LIN {X 0,Y 269.513,Z 759.84,A -85,B 0,C 180,E1 -29388.002,E2 -29388.002} C_VEL
LIN {X 0,Y 275.848,Z 764.701,A -85,B 0,C 180,E1 -29390.437,E2 -29390.437} C_VEL
LIN {X 0,Y 281.948,Z 769.462,A -85,B 0,C 180,E1 -29392.905,E2 -29392.905} C_VEL
LIN {X 0,Y 289.279,Z 774.875,A -85,B 0,C 180,E1 -29396.029,E2 -29396.029} C_VEL
LIN {X 0,Y 294.079,Z 778.705,A -85,B 0,C 180,E1 -29398.281,E2 -29398.281} C_VEL
LIN {X 0,Y 298.716,Z 782.114,A -85,B 0,C 180,E1 -29400.517,E2 -29400.517} C_VEL
LIN {X 0,Y 303.536,Z 785.554,A -85,B 0,C 180,E1 -29402.995,E2 -29402.995} C_VEL
LIN {X 0,Y 308.5,Z 789.254,A -85,B 0,C 180,E1 -29405.792,E2 -29405.792} C_VEL
LIN {X 0,Y 311.598,Z 791.295,A -85,B 0,C 180,E1 -29407.628,E2 -29407.628} C_VEL
LIN {X 0,Y 314.778,Z 793.373,A -85,B 0,C 180,E1 -29409.672,E2 -29409.672} C_VEL
LIN {X 0,Y 317.869,Z 795.742,A -85,B 0,C 180,E1 -29411.969,E2 -29411.969} C_VEL
LIN {X 0,Y 321.084,Z 798.198,A -85,B 0,C 180,E1 -29414.772,E2 -29414.772} C_VEL
LIN {X 0,Y 323.911,Z 800.084,A -85,B 0,C 180,E1 -29417.519,E2 -29417.519} C_VEL
LIN {X 0,Y 326.293,Z 801.22,A -85,B 0,C 180,E1 -29420.078,E2 -29420.078} C_VEL
LIN {X 0,Y 328.105,Z 802.015,A -85,B 0,C 180,E1 -29422.616,E2 -29422.616} C_VEL
LIN {X 0,Y 329.27,Z 802.725,A -85,B 0,C 180,E1 -29425.102,E2 -29425.102} C_VEL
LIN {X 0,Y 330.146,Z 802.967,A -85,B 0,C 180,E1 -29427.56,E2 -29427.56} C_VEL
LIN {X 0,Y 330.328,Z 803.159,A -85,B 0,C 180,E1 -29430,E2 -29430} C_VEL
LIN {X 0,Y 330.117,Z 802.967,A -85,B 0,C 180,E1 -29432.44,E2 -29432.44} C_VEL
LIN {X 0,Y 329.312,Z 802.689,A -85,B 0,C 180,E1 -29434.897,E2 -29434.897} C_VEL
LIN {X 0,Y 328.123,Z 802.039,A -85,B 0,C 180,E1 -29437.383,E2 -29437.383} C_VEL
LIN {X 0,Y 326.265,Z 801.233,A -85,B 0,C 180,E1 -29439.923,E2 -29439.923} C_VEL
LIN {X 0,Y 323.871,Z 800.004,A -85,B 0,C 180,E1 -29442.533,E2 -29442.533} C_VEL
LIN {X 0,Y 320.809,Z 798.053,A -85,B 0,C 180,E1 -29445.442,E2 -29445.442} C_VEL
LIN {X 0,Y 317.814,Z 795.774,A -85,B 0,C 180,E1 -29448.034,E2 -29448.034} C_VEL
LIN {X 0,Y 314.765,Z 793.38,A -85,B 0,C 180,E1 -29450.322,E2 -29450.322} C_VEL
LIN {X 0,Y 311.247,Z 791.126,A -85,B 0,C 180,E1 -29452.573,E2 -29452.573} C_VEL
LIN {X 0,Y 305.558,Z 787.096,A -85,B 0,C 180,E1 -29455.913,E2 -29455.913} C_VEL
LIN {X 0,Y 300.069,Z 782.993,A -85,B 0,C 180,E1 -29458.828,E2 -29458.828} C_VEL
LIN {X 0,Y 294.071,Z 778.695,A -85,B 0,C 180,E1 -29461.72,E2 -29461.72} C_VEL
LIN {X 0,Y 288.811,Z 774.531,A -85,B 0,C 180,E1 -29464.172,E2 -29464.172} C_VEL
LIN {X 0,Y 281.952,Z 769.478,A -85,B 0,C 180,E1 -29467.096,E2 -29467.096} C_VEL
LIN {X 0,Y 275.891,Z 764.765,A -85,B 0,C 180,E1 -29469.556,E2 -29469.556} C_VEL
LIN {X 0,Y 269.548,Z 759.774,A -85,B 0,C 180,E1 -29472.006,E2 -29472.006} C_VEL
LIN {X 0,Y 260.297,Z 752.713,A -85,B 0,C 180,E1 -29475.413,E2 -29475.413} C_VEL
LIN {X 0,Y 246.486,Z 741.482,A -85,B 0,C 180,E1 -29481.151,E2 -29481.151} C_VEL
LIN {X 0,Y 233.507,Z 728.442,A -85,B 0,C 180,E1 -29488.217,E2 -29488.217} C_VEL
LIN {X 0,Y 225.035,Z 716.362,A -85,B 0,C 180,E1 -29494.682,E2 -29494.682} C_VEL
LIN {X 0,Y 219.674,Z 703.721,A -85,B 0,C 180,E1 -29500.918,E2 -29500.918} C_VEL
LIN {X 0,Y 216.948,Z 692.283,A -85,B 0,C 180,E1 -29506.06,E2 -29506.06} C_VEL
LIN {X 0,Y 215.599,Z 681.886,A -85,B 0,C 180,E1 -29510.507,E2 -29510.507} C_VEL
LIN {X 0,Y 214.994,Z 678.195,A -85,B 0,C 180,E1 -29512.664,E2 -29512.664} C_VEL
LIN {X 0,Y 214.461,Z 674.849,A -85,B 0,C 180,E1 -29515.412,E2 -29515.412} C_VEL
LIN {X 0,Y 214.209,Z 673.133,A -85,B 0,C 180,E1 -29517.65,E2 -29517.65} C_VEL
LIN {X 0,Y 214.12,Z 672.763,A -85,B 0,C 180,E1 -29520.476,E2 -29520.476} C_VEL
LIN {X 0,Y 211.138,Z 691.221,A -85,B 0,C 180,E1 -29520.708,E2 -29520.708} C_VEL
LIN {X 0,Y 207.685,Z 705.637,A -85,B 0,C 180,E1 -29520.907,E2 -29520.907} C_VEL
LIN {X 0,Y 203.406,Z 719.374,A -85,B 0,C 180,E1 -29521.115,E2 -29521.115} C_VEL
LIN {X 0,Y 198.594,Z 731.963,A -85,B 0,C 180,E1 -29521.377,E2 -29521.377} C_VEL
LIN {X 0,Y 193.349,Z 743.558,A -85,B 0,C 180,E1 -29521.688,E2 -29521.688} C_VEL
LIN {X 0,Y 186.937,Z 755.704,A -85,B 0,C 180,E1 -29522.084,E2 -29522.084} C_VEL
LIN {X 0,Y 179.399,Z 768.002,A -85,B 0,C 180,E1 -29522.63,E2 -29522.63} C_VEL
LIN {X 0,Y 171.572,Z 779.121,A -85,B 0,C 180,E1 -29523.206,E2 -29523.206} C_VEL
LIN {X 0,Y 162.906,Z 789.948,A -85,B 0,C 180,E1 -29523.954,E2 -29523.954} C_VEL
LIN {X 0,Y 153.235,Z 800.571,A -85,B 0,C 180,E1 -29524.879,E2 -29524.879} C_VEL
LIN {X 0,Y 144.516,Z 809.109,A -85,B 0,C 180,E1 -29525.913,E2 -29525.913} C_VEL
LIN {X 0,Y 134.582,Z 817.767,A -85,B 0,C 180,E1 -29527.172,E2 -29527.172} C_VEL
LIN {X 0,Y 124.423,Z 825.65,A -85,B 0,C 180,E1 -29528.714,E2 -29528.714} C_VEL
LIN {X 0,Y 113.699,Z 833.04,A -85,B 0,C 180,E1 -29530.687,E2 -29530.687} C_VEL
LIN {X 0,Y 101.25,Z 840.568,A -85,B 0,C 180,E1 -29533.65,E2 -29533.65} C_VEL
LIN {X 0,Y 91.621,Z 845.7,A -85,B 0,C 180,E1 -29536.501,E2 -29536.501} C_VEL
LIN {X 0,Y 79.232,Z 851.465,A -85,B 0,C 180,E1 -29541.354,E2 -29541.354} C_VEL
LIN {X 0,Y 70.415,Z 855.088,A -85,B 0,C 180,E1 -29546.071,E2 -29546.071} C_VEL
LIN {X 0,Y 59.652,Z 858.961,A -85,B 0,C 180,E1 -29554.442,E2 -29554.442} C_VEL
LIN {X 0,Y 50.575,Z 861.84,A -85,B 0,C 180,E1 -29565.99,E2 -29565.99} C_VEL
LIN {X 0,Y 44.024,Z 863.755,A -85,B 0,C 180,E1 -29581.386,E2 -29581.386} C_VEL
LIN {X 0,Y 42.132,Z 864.451,A -85,B 0,C 180,E1 -29590.512,E2 -29590.512} C_VEL
LIN {X 0,Y 41.238,Z 864.959,A -85,B 0,C 180,E1 -29610,E2 -29610} C_VEL
LIN {X 0,Y 42.12,Z 864.45,A -85,B 0,C 180,E1 -29629.494,E2 -29629.494} C_VEL
LIN {X 0,Y 46.907,Z 862.99,A -85,B 0,C 180,E1 -29646.82,E2 -29646.82} C_VEL
LIN {X 0,Y 54.867,Z 860.576,A -85,B 0,C 180,E1 -29660.223,E2 -29660.223} C_VEL
LIN {X 0,Y 67.596,Z 856.132,A -85,B 0,C 180,E1 -29672.096,E2 -29672.096} C_VEL
LIN {X 0,Y 76.226,Z 852.753,A -85,B 0,C 180,E1 -29677.216,E2 -29677.216} C_VEL
LIN {X 0,Y 88.465,Z 847.245,A -85,B 0,C 180,E1 -29682.422,E2 -29682.422} C_VEL
LIN {X 0,Y 98.02,Z 842.385,A -85,B 0,C 180,E1 -29685.448,E2 -29685.448} C_VEL
LIN {X 0,Y 110.913,Z 834.823,A -85,B 0,C 180,E1 -29688.675,E2 -29688.675} C_VEL
LIN {X 0,Y 121.061,Z 828.065,A -85,B 0,C 180,E1 -29690.711,E2 -29690.711} C_VEL
LIN {X 0,Y 131.176,Z 820.52,A -85,B 0,C 180,E1 -29692.371,E2 -29692.371} C_VEL
LIN {X 0,Y 141.415,Z 811.951,A -85,B 0,C 180,E1 -29693.685,E2 -29693.685} C_VEL
LIN {X 0,Y 151.346,Z 802.524,A -85,B 0,C 180,E1 -29694.899,E2 -29694.899} C_VEL
LIN {X 0,Y 161.169,Z 791.956,A -85,B 0,C 180,E1 -29695.927,E2 -29695.927} C_VEL
LIN {X 0,Y 169.832,Z 781.404,A -85,B 0,C 180,E1 -29696.676,E2 -29696.676} C_VEL
LIN {X 0,Y 177.659,Z 770.609,A -85,B 0,C 180,E1 -29697.242,E2 -29697.242} C_VEL
LIN {X 0,Y 185.055,Z 758.937,A -85,B 0,C 180,E1 -29697.793,E2 -29697.793} C_VEL
LIN {X 0,Y 191.601,Z 747.036,A -85,B 0,C 180,E1 -29698.219,E2 -29698.219} C_VEL
LIN {X 0,Y 197.282,Z 735.038,A -85,B 0,C 180,E1 -29698.545,E2 -29698.545} C_VEL
LIN {X 0,Y 202.532,Z 721.843,A -85,B 0,C 180,E1 -29698.826,E2 -29698.826} C_VEL
LIN {X 0,Y 206.767,Z 708.849,A -85,B 0,C 180,E1 -29699.043,E2 -29699.043} C_VEL
LIN {X 0,Y 210.248,Z 695.285,A -85,B 0,C 180,E1 -29699.228,E2 -29699.228} C_VEL
LIN {X 0,Y 212.638,Z 682.821,A -85,B 0,C 180,E1 -29699.413,E2 -29699.413} C_VEL
LIN {X 0,Y 214.121,Z 672.732,A -85,B 0,C 180,E1 -29699.584,E2 -29699.584} C_VEL
LIN {X 0,Y 214.238,Z 673.333,A -85,B 0,C 180,E1 -29702.702,E2 -29702.702} C_VEL
LIN {X 0,Y 214.62,Z 675.963,A -85,B 0,C 180,E1 -29705.637,E2 -29705.637} C_VEL
LIN {X 0,Y 215.251,Z 679.856,A -85,B 0,C 180,E1 -29708.419,E2 -29708.419} C_VEL
LIN {X 0,Y 215.918,Z 684.51,A -85,B 0,C 180,E1 -29710.668,E2 -29710.668} C_VEL
LIN {X 0,Y 216.528,Z 689.348,A -85,B 0,C 180,E1 -29712.698,E2 -29712.698} C_VEL
LIN {X 0,Y 216.824,Z 691.412,A -85,B 0,C 180,E1 -29713.574,E2 -29713.574} C_VEL
LIN {X 0,Y 217.026,Z 695.327,A -85,B 0,C 180,E1 -29714.74,E2 -29714.74} C_VEL
LIN {X 0,Y 216.849,Z 707.033,A -85,B 0,C 180,E1 -29717.584,E2 -29717.584} C_VEL
LIN {X 0,Y 217.221,Z 710.631,A -85,B 0,C 180,E1 -29718.824,E2 -29718.824} C_VEL
LIN {X 0,Y 222.051,Z 722.799,A -85,B 0,C 180,E1 -29725.068,E2 -29725.068} C_VEL
LIN {X 0,Y 230.801,Z 735.633,A -85,B 0,C 180,E1 -29732.2,E2 -29732.2} C_VEL
LIN {X 0,Y 245.264,Z 749.741,A -85,B 0,C 180,E1 -29740.145,E2 -29740.145} C_VEL
LIN {X 0,Y 257.353,Z 759.43,A -85,B 0,C 180,E1 -29745.236,E2 -29745.236} C_VEL
LIN {X 0,Y 264.757,Z 765.09,A -85,B 0,C 180,E1 -29748.009,E2 -29748.009} C_VEL
LIN {X 0,Y 271.997,Z 770.662,A -85,B 0,C 180,E1 -29750.818,E2 -29750.818} C_VEL
LIN {X 0,Y 277.29,Z 774.8,A -85,B 0,C 180,E1 -29752.973,E2 -29752.973} C_VEL
LIN {X 0,Y 284.234,Z 779.942,A -85,B 0,C 180,E1 -29755.926,E2 -29755.926} C_VEL
LIN {X 0,Y 289.243,Z 783.893,A -85,B 0,C 180,E1 -29758.257,E2 -29758.257} C_VEL
LIN {X 0,Y 294.145,Z 787.523,A -85,B 0,C 180,E1 -29760.628,E2 -29760.628} C_VEL
LIN {X 0,Y 299.172,Z 791.122,A -85,B 0,C 180,E1 -29763.21,E2 -29763.21} C_VEL
LIN {X 0,Y 302.926,Z 793.936,A -85,B 0,C 180,E1 -29765.317,E2 -29765.317} C_VEL
LIN {X 0,Y 305.799,Z 795.921,A -85,B 0,C 180,E1 -29767.002,E2 -29767.002} C_VEL
LIN {X 0,Y 308.863,Z 797.869,A -85,B 0,C 180,E1 -29768.894,E2 -29768.894} C_VEL
LIN {X 0,Y 312.723,Z 800.732,A -85,B 0,C 180,E1 -29771.662,E2 -29771.662} C_VEL
LIN {X 0,Y 316.06,Z 803.297,A -85,B 0,C 180,E1 -29774.524,E2 -29774.524} C_VEL
LIN {X 0,Y 318.94,Z 805.266,A -85,B 0,C 180,E1 -29777.27,E2 -29777.27} C_VEL
LIN {X 0,Y 321.428,Z 806.457,A -85,B 0,C 180,E1 -29779.926,E2 -29779.926} C_VEL
LIN {X 0,Y 323.337,Z 807.296,A -85,B 0,C 180,E1 -29782.507,E2 -29782.507} C_VEL
LIN {X 0,Y 324.551,Z 808.043,A -85,B 0,C 180,E1 -29785.031,E2 -29785.031} C_VEL
LIN {X 0,Y 325.474,Z 808.31,A -85,B 0,C 180,E1 -29787.525,E2 -29787.525} C_VEL
LIN {X 0,Y 325.699,Z 808.396,A -85,B 0,C 180,E1 -29788.764,E2 -29788.764} C_VEL
LIN {X 0,Y 325.626,Z 808.426,A -85,B 0,C 180,E1 -29791.237,E2 -29791.237} C_VEL
LIN {X 0,Y 325.034,Z 808.243,A -85,B 0,C 180,E1 -29793.719,E2 -29793.719} C_VEL
LIN {X 0,Y 324.061,Z 807.683,A -85,B 0,C 180,E1 -29796.225,E2 -29796.225} C_VEL
LIN {X 0,Y 322.442,Z 806.929,A -85,B 0,C 180,E1 -29798.776,E2 -29798.776} C_VEL
LIN {X 0,Y 320.245,Z 805.898,A -85,B 0,C 180,E1 -29801.391,E2 -29801.391} C_VEL
LIN {X 0,Y 317.542,Z 804.326,A -85,B 0,C 180,E1 -29804.09,E2 -29804.09} C_VEL
LIN {X 0,Y 314.395,Z 802.115,A -85,B 0,C 180,E1 -29806.894,E2 -29806.894} C_VEL
LIN {X 0,Y 311.99,Z 800.188,A -85,B 0,C 180,E1 -29808.898,E2 -29808.898} C_VEL
LIN {X 0,Y 308.435,Z 797.598,A -85,B 0,C 180,E1 -29811.381,E2 -29811.381} C_VEL
LIN {X 0,Y 305.606,Z 795.851,A -85,B 0,C 180,E1 -29813.094,E2 -29813.094} C_VEL
LIN {X 0,Y 299.862,Z 791.627,A -85,B 0,C 180,E1 -29816.443,E2 -29816.443} C_VEL
LIN {X 0,Y 294.191,Z 787.506,A -85,B 0,C 180,E1 -29819.37,E2 -29819.37} C_VEL
LIN {X 0,Y 289.247,Z 783.903,A -85,B 0,C 180,E1 -29821.744,E2 -29821.744} C_VEL
LIN {X 0,Y 284.24,Z 779.944,A -85,B 0,C 180,E1 -29824.076,E2 -29824.076} C_VEL
LIN {X 0,Y 279.029,Z 776.124,A -85,B 0,C 180,E1 -29826.295,E2 -29826.295} C_VEL
LIN {X 0,Y 275.596,Z 773.373,A -85,B 0,C 180,E1 -29827.766,E2 -29827.766} C_VEL
LIN {X 0,Y 268.399,Z 767.914,A -85,B 0,C 180,E1 -29830.593,E2 -29830.593} C_VEL
LIN {X 0,Y 262.635,Z 763.36,A -85,B 0,C 180,E1 -29832.785,E2 -29832.785} C_VEL
LIN {X 0,Y 250.326,Z 753.803,A -85,B 0,C 180,E1 -29837.639,E2 -29837.639} C_VEL
LIN {X 0,Y 234.708,Z 740.007,A -85,B 0,C 180,E1 -29845.325,E2 -29845.325} C_VEL
LIN {X 0,Y 225.105,Z 728.004,A -85,B 0,C 180,E1 -29852.076,E2 -29852.076} C_VEL
LIN {X 0,Y 219.774,Z 718.027,A -85,B 0,C 180,E1 -29857.435,E2 -29857.435} C_VEL
LIN {X 0,Y 216.366,Z 707.28,A -85,B 0,C 180,E1 -29862.759,E2 -29862.759} C_VEL
LIN {X 0,Y 214.647,Z 696.607,A -85,B 0,C 180,E1 -29867.605,E2 -29867.605} C_VEL
LIN {X 0,Y 213.992,Z 687.722,A -85,B 0,C 180,E1 -29871.531,E2 -29871.531} C_VEL
LIN {X 0,Y 213.696,Z 684.84,A -85,B 0,C 180,E1 -29873.242,E2 -29873.242} C_VEL
LIN {X 0,Y 213.348,Z 681.75,A -85,B 0,C 180,E1 -29875.741,E2 -29875.741} C_VEL
LIN {X 0,Y 213.161,Z 680.078,A -85,B 0,C 180,E1 -29878.111,E2 -29878.111} C_VEL
LIN {X 0,Y 213.13,Z 679.974,A -85,B 0,C 180,E1 -29878.628,E2 -29878.628} C_VEL
LIN {X 0,Y 210.458,Z 694.251,A -85,B 0,C 180,E1 -29878.816,E2 -29878.816} C_VEL
LIN {X 0,Y 206.952,Z 708.017,A -85,B 0,C 180,E1 -29878.971,E2 -29878.971} C_VEL
LIN {X 0,Y 202.511,Z 721.639,A -85,B 0,C 180,E1 -29879.156,E2 -29879.156} C_VEL
LIN {X 0,Y 197.23,Z 734.836,A -85,B 0,C 180,E1 -29879.381,E2 -29879.381} C_VEL
LIN {X 0,Y 190.633,Z 748.57,A -85,B 0,C 180,E1 -29879.697,E2 -29879.697} C_VEL
LIN {X 0,Y 180.968,Z 765.188,A -85,B 0,C 180,E1 -29880.256,E2 -29880.256} C_VEL
LIN {X 0,Y 172.197,Z 777.773,A -85,B 0,C 180,E1 -29880.752,E2 -29880.752} C_VEL
LIN {X 0,Y 163.445,Z 788.736,A -85,B 0,C 180,E1 -29881.387,E2 -29881.387} C_VEL
LIN {X 0,Y 154.71,Z 798.412,A -85,B 0,C 180,E1 -29882.033,E2 -29882.033} C_VEL
LIN {X 0,Y 145.707,Z 807.315,A -85,B 0,C 180,E1 -29882.877,E2 -29882.877} C_VEL
LIN {X 0,Y 135.611,Z 816.181,A -85,B 0,C 180,E1 -29883.966,E2 -29883.966} C_VEL
LIN {X 0,Y 123.537,Z 825.437,A -85,B 0,C 180,E1 -29885.407,E2 -29885.407} C_VEL
LIN {X 0,Y 113.281,Z 832.397,A -85,B 0,C 180,E1 -29886.965,E2 -29886.965} C_VEL
LIN {X 0,Y 103.144,Z 838.537,A -85,B 0,C 180,E1 -29888.895,E2 -29888.895} C_VEL
LIN {X 0,Y 89.836,Z 845.486,A -85,B 0,C 180,E1 -29892.076,E2 -29892.076} C_VEL
LIN {X 0,Y 79.188,Z 850.32,A -85,B 0,C 180,E1 -29895.442,E2 -29895.442} C_VEL
LIN {X 0,Y 67.558,Z 854.875,A -85,B 0,C 180,E1 -29900.571,E2 -29900.571} C_VEL
LIN {X 0,Y 55.889,Z 858.747,A -85,B 0,C 180,E1 -29908.331,E2 -29908.331} C_VEL
LIN {X 0,Y 49.655,Z 860.644,A -85,B 0,C 180,E1 -29914.484,E2 -29914.484} C_VEL
LIN {X 0,Y 41.387,Z 862.778,A -85,B 0,C 180,E1 -29927.217,E2 -29927.217} C_VEL
LIN {X 0,Y 35.444,Z 864.239,A -85,B 0,C 180,E1 -29946.637,E2 -29946.637} C_VEL
LIN {X 0,Y 34.113,Z 864.748,A -85,B 0,C 180,E1 -29970,E2 -29970} C_VEL
LIN {X 0,Y 35.435,Z 864.238,A -85,B 0,C 180,E1 -29993.37,E2 -29993.37} C_VEL
LIN {X 0,Y 41.386,Z 862.778,A -85,B 0,C 180,E1 -30012.785,E2 -30012.785} C_VEL
LIN {X 0,Y 50.551,Z 860.362,A -85,B 0,C 180,E1 -30026.527,E2 -30026.527} C_VEL
LIN {X 0,Y 64.534,Z 855.919,A -85,B 0,C 180,E1 -30037.767,E2 -30037.767} C_VEL
LIN {X 0,Y 73.73,Z 852.54,A -85,B 0,C 180,E1 -30042.399,E2 -30042.399} C_VEL
LIN {X 0,Y 86.56,Z 847.032,A -85,B 0,C 180,E1 -30046.978,E2 -30046.978} C_VEL
LIN {X 0,Y 96.457,Z 842.171,A -85,B 0,C 180,E1 -30049.61,E2 -30049.61} C_VEL
LIN {X 0,Y 109.237,Z 834.915,A -85,B 0,C 180,E1 -30052.278,E2 -30052.278} C_VEL
LIN {X 0,Y 120.108,Z 827.852,A -85,B 0,C 180,E1 -30054.109,E2 -30054.109} C_VEL
LIN {X 0,Y 130.416,Z 820.307,A -85,B 0,C 180,E1 -30055.504,E2 -30055.504} C_VEL
LIN {X 0,Y 140.806,Z 811.74,A -85,B 0,C 180,E1 -30056.587,E2 -30056.587} C_VEL
LIN {X 0,Y 151.225,Z 801.959,A -85,B 0,C 180,E1 -30057.652,E2 -30057.652} C_VEL
LIN {X 0,Y 160.819,Z 791.748,A -85,B 0,C 180,E1 -30058.464,E2 -30058.464} C_VEL
LIN {X 0,Y 169.568,Z 781.199,A -85,B 0,C 180,E1 -30059.076,E2 -30059.076} C_VEL
LIN {X 0,Y 177.458,Z 770.402,A -85,B 0,C 180,E1 -30059.545,E2 -30059.545} C_VEL
LIN {X 0,Y 184.757,Z 759.006,A -85,B 0,C 180,E1 -30060,E2 -30060} C_VEL
LIN {X 0,Y 191.512,Z 746.83,A -85,B 0,C 180,E1 -30060.348,E2 -30060.348} C_VEL
LIN {X 0,Y 197.23,Z 734.836,A -85,B 0,C 180,E1 -30060.618,E2 -30060.618} C_VEL
LIN {X 0,Y 202.511,Z 721.64,A -85,B 0,C 180,E1 -30060.836,E2 -30060.836} C_VEL
LIN {X 0,Y 206.73,Z 708.788,A -85,B 0,C 180,E1 -30061.01,E2 -30061.01} C_VEL
LIN {X 0,Y 210.233,Z 695.271,A -85,B 0,C 180,E1 -30061.164,E2 -30061.164} C_VEL
LIN {X 0,Y 212.782,Z 681.98,A -85,B 0,C 180,E1 -30061.333,E2 -30061.333} C_VEL
LIN {X 0,Y 213.102,Z 679.928,A -85,B 0,C 180,E1 -30061.372,E2 -30061.372} C_VEL
LIN {X 0,Y 213.183,Z 680.8,A -85,B 0,C 180,E1 -30063.07,E2 -30063.07} C_VEL
LIN {X 0,Y 213.486,Z 683.323,A -85,B 0,C 180,E1 -30065.667,E2 -30065.667} C_VEL
LIN {X 0,Y 213.912,Z 686.53,A -85,B 0,C 180,E1 -30067.848,E2 -30067.848} C_VEL
LIN {X 0,Y 214.208,Z 691.624,A -85,B 0,C 180,E1 -30070.252,E2 -30070.252} C_VEL
LIN {X 0,Y 215.674,Z 704.072,A -85,B 0,C 180,E1 -30075.716,E2 -30075.716} C_VEL
LIN {X 0,Y 217.221,Z 710.631,A -85,B 0,C 180,E1 -30078.824,E2 -30078.824} C_VEL
LIN {X 0,Y 217.704,Z 714.076,A -85,B 0,C 180,E1 -30080.089,E2 -30080.089} C_VEL
LIN {X 0,Y 218.379,Z 727.051,A -85,B 0,C 180,E1 -30084.004,E2 -30084.004} C_VEL
LIN {X 0,Y 219.25,Z 729.971,A -85,B 0,C 180,E1 -30085.317,E2 -30085.317} C_VEL
LIN {X 0,Y 226.67,Z 741.194,A -85,B 0,C 180,E1 -30091.809,E2 -30091.809} C_VEL
LIN {X 0,Y 239.104,Z 753.74,A -85,B 0,C 180,E1 -30099.193,E2 -30099.193} C_VEL
LIN {X 0,Y 250.711,Z 763.192,A -85,B 0,C 180,E1 -30104.491,E2 -30104.491} C_VEL
LIN {X 0,Y 259.783,Z 770.151,A -85,B 0,C 180,E1 -30108.07,E2 -30108.07} C_VEL
LIN {X 0,Y 266.852,Z 775.583,A -85,B 0,C 180,E1 -30110.797,E2 -30110.797} C_VEL
LIN {X 0,Y 274.503,Z 781.5,A -85,B 0,C 180,E1 -30113.925,E2 -30113.925} C_VEL
LIN {X 0,Y 280.674,Z 786.071,A -85,B 0,C 180,E1 -30116.574,E2 -30116.574} C_VEL
LIN {X 0,Y 286.252,Z 790.444,A -85,B 0,C 180,E1 -30119.238,E2 -30119.238} C_VEL
LIN {X 0,Y 291.295,Z 794.06,A -85,B 0,C 180,E1 -30121.715,E2 -30121.715} C_VEL
LIN {X 0,Y 296.224,Z 797.714,A -85,B 0,C 180,E1 -30124.362,E2 -30124.362} C_VEL
LIN {X 0,Y 299.987,Z 800.438,A -85,B 0,C 180,E1 -30126.53,E2 -30126.53} C_VEL
LIN {X 0,Y 305.214,Z 803.872,A -85,B 0,C 180,E1 -30129.794,E2 -30129.794} C_VEL
LIN {X 0,Y 307.291,Z 805.44,A -85,B 0,C 180,E1 -30131.326,E2 -30131.326} C_VEL
LIN {X 0,Y 310.769,Z 808.143,A -85,B 0,C 180,E1 -30134.254,E2 -30134.254} C_VEL
LIN {X 0,Y 313.736,Z 810.196,A -85,B 0,C 180,E1 -30137.056,E2 -30137.056} C_VEL
LIN {X 0,Y 316.301,Z 811.474,A -85,B 0,C 180,E1 -30139.761,E2 -30139.761} C_VEL
LIN {X 0,Y 318.33,Z 812.356,A -85,B 0,C 180,E1 -30142.388,E2 -30142.388} C_VEL
LIN {X 0,Y 319.622,Z 813.123,A -85,B 0,C 180,E1 -30144.954,E2 -30144.954} C_VEL
LIN {X 0,Y 320.566,Z 813.433,A -85,B 0,C 180,E1 -30147.487,E2 -30147.487} C_VEL
LIN {X 0,Y 320.806,Z 813.51,A -85,B 0,C 180,E1 -30148.745,E2 -30148.745} C_VEL
LIN {X 0,Y 320.716,Z 813.556,A -85,B 0,C 180,E1 -30151.256,E2 -30151.256} C_VEL
LIN {X 0,Y 320.539,Z 813.431,A -85,B 0,C 180,E1 -30152.513,E2 -30152.513} C_VEL
LIN {X 0,Y 319.665,Z 813.099,A -85,B 0,C 180,E1 -30155.045,E2 -30155.045} C_VEL
LIN {X 0,Y 318.33,Z 812.397,A -85,B 0,C 180,E1 -30157.612,E2 -30157.612} C_VEL
LIN {X 0,Y 316.288,Z 811.464,A -85,B 0,C 180,E1 -30160.239,E2 -30160.239} C_VEL
LIN {X 0,Y 313.763,Z 810.131,A -85,B 0,C 180,E1 -30162.943,E2 -30162.943} C_VEL
LIN {X 0,Y 310.723,Z 808.146,A -85,B 0,C 180,E1 -30165.748,E2 -30165.748} C_VEL
LIN {X 0,Y 307.272,Z 805.442,A -85,B 0,C 180,E1 -30168.675,E2 -30168.675} C_VEL
LIN {X 0,Y 305.219,Z 803.889,A -85,B 0,C 180,E1 -30170.205,E2 -30170.205} C_VEL
LIN {X 0,Y 302.732,Z 802.227,A -85,B 0,C 180,E1 -30171.804,E2 -30171.804} C_VEL
LIN {X 0,Y 299.467,Z 800.127,A -85,B 0,C 180,E1 -30173.758,E2 -30173.758} C_VEL
LIN {X 0,Y 293.734,Z 795.821,A -85,B 0,C 180,E1 -30177.039,E2 -30177.039} C_VEL
LIN {X 0,Y 289.667,Z 792.874,A -85,B 0,C 180,E1 -30179.14,E2 -30179.14} C_VEL
LIN {X 0,Y 282.904,Z 787.825,A -85,B 0,C 180,E1 -30182.368,E2 -30182.368} C_VEL
LIN {X 0,Y 277.992,Z 784.082,A -85,B 0,C 180,E1 -30184.584,E2 -30184.584} C_VEL
LIN {X 0,Y 271.434,Z 779.106,A -85,B 0,C 180,E1 -30187.357,E2 -30187.357} C_VEL
LIN {X 0,Y 265.294,Z 774.465,A -85,B 0,C 180,E1 -30189.804,E2 -30189.804} C_VEL
LIN {X 0,Y 257.977,Z 768.668,A -85,B 0,C 180,E1 -30192.647,E2 -30192.647} C_VEL
LIN {X 0,Y 245.577,Z 759.11,A -85,B 0,C 180,E1 -30197.738,E2 -30197.738} C_VEL
LIN {X 0,Y 230.449,Z 745.541,A -85,B 0,C 180,E1 -30205.653,E2 -30205.653} C_VEL
LIN {X 0,Y 220.993,Z 733.049,A -85,B 0,C 180,E1 -30212.927,E2 -30212.927} C_VEL
LIN {X 0,Y 216.401,Z 723.37,A -85,B 0,C 180,E1 -30218.308,E2 -30218.308} C_VEL
LIN {X 0,Y 213.592,Z 712.701,A -85,B 0,C 180,E1 -30223.759,E2 -30223.759} C_VEL
LIN {X 0,Y 212.397,Z 700.51,A -85,B 0,C 180,E1 -30229.379,E2 -30229.379} C_VEL
LIN {X 0,Y 212.235,Z 693.67,A -85,B 0,C 180,E1 -30232.461,E2 -30232.461} C_VEL
LIN {X 0,Y 212.142,Z 691.135,A -85,B 0,C 180,E1 -30234.035,E2 -30234.035} C_VEL
LIN {X 0,Y 212.057,Z 688.368,A -85,B 0,C 180,E1 -30236.414,E2 -30236.414} C_VEL
LIN {X 0,Y 212.038,Z 688.086,A -85,B 0,C 180,E1 -30236.797,E2 -30236.797} C_VEL
LIN {X 0,Y 208.044,Z 704.898,A -85,B 0,C 180,E1 -30236.986,E2 -30236.986} C_VEL
LIN {X 0,Y 203.626,Z 718.969,A -85,B 0,C 180,E1 -30237.117,E2 -30237.117} C_VEL
LIN {X 0,Y 198.76,Z 731.56,A -85,B 0,C 180,E1 -30237.279,E2 -30237.279} C_VEL
LIN {X 0,Y 193.455,Z 743.145,A -85,B 0,C 180,E1 -30237.464,E2 -30237.464} C_VEL
LIN {X 0,Y 187.001,Z 755.229,A -85,B 0,C 180,E1 -30237.719,E2 -30237.719} C_VEL
LIN {X 0,Y 179.311,Z 767.588,A -85,B 0,C 180,E1 -30238.077,E2 -30238.077} C_VEL
LIN {X 0,Y 171.368,Z 778.709,A -85,B 0,C 180,E1 -30238.422,E2 -30238.422} C_VEL
LIN {X 0,Y 162.547,Z 789.533,A -85,B 0,C 180,E1 -30238.929,E2 -30238.929} C_VEL
LIN {X 0,Y 152.861,Z 799.977,A -85,B 0,C 180,E1 -30239.493,E2 -30239.493} C_VEL
LIN {X 0,Y 143.041,Z 809.317,A -85,B 0,C 180,E1 -30240.25,E2 -30240.25} C_VEL
LIN {X 0,Y 133.552,Z 817.349,A -85,B 0,C 180,E1 -30241.076,E2 -30241.076} C_VEL
LIN {X 0,Y 123.067,Z 825.227,A -85,B 0,C 180,E1 -30242.071,E2 -30242.071} C_VEL
LIN {X 0,Y 112.635,Z 832.186,A -85,B 0,C 180,E1 -30243.326,E2 -30243.326} C_VEL
LIN {X 0,Y 102.276,Z 838.324,A -85,B 0,C 180,E1 -30244.89,E2 -30244.89} C_VEL
LIN {X 0,Y 88.608,Z 845.273,A -85,B 0,C 180,E1 -30247.509,E2 -30247.509} C_VEL
LIN {X 0,Y 76.671,Z 850.458,A -85,B 0,C 180,E1 -30250.565,E2 -30250.565} C_VEL
LIN {X 0,Y 65.368,Z 854.661,A -85,B 0,C 180,E1 -30254.624,E2 -30254.624} C_VEL
LIN {X 0,Y 52.847,Z 858.534,A -85,B 0,C 180,E1 -30261.425,E2 -30261.425} C_VEL
LIN {X 0,Y 41.443,Z 861.414,A -85,B 0,C 180,E1 -30272.018,E2 -30272.018} C_VEL
LIN {X 0,Y 36.45,Z 862.566,A -85,B 0,C 180,E1 -30279.536,E2 -30279.536} C_VEL
LIN {X 0,Y 29.004,Z 864.027,A -85,B 0,C 180,E1 -30301.012,E2 -30301.012} C_VEL
LIN {X 0,Y 27.001,Z 864.538,A -85,B 0,C 180,E1 -30330,E2 -30330} C_VEL
LIN {X 0,Y 28.996,Z 864.026,A -85,B 0,C 180,E1 -30358.996,E2 -30358.996} C_VEL
LIN {X 0,Y 36.449,Z 862.566,A -85,B 0,C 180,E1 -30380.466,E2 -30380.466} C_VEL
LIN {X 0,Y 46.962,Z 860.149,A -85,B 0,C 180,E1 -30393.884,E2 -30393.884} C_VEL
LIN {X 0,Y 62.167,Z 855.706,A -85,B 0,C 180,E1 -30403.924,E2 -30403.924} C_VEL
LIN {X 0,Y 71.878,Z 852.326,A -85,B 0,C 180,E1 -30407.889,E2 -30407.889} C_VEL
LIN {X 0,Y 85.224,Z 846.819,A -85,B 0,C 180,E1 -30411.711,E2 -30411.711} C_VEL
LIN {X 0,Y 95.421,Z 841.958,A -85,B 0,C 180,E1 -30413.871,E2 -30413.871} C_VEL
LIN {X 0,Y 109.172,Z 834.295,A -85,B 0,C 180,E1 -30416.158,E2 -30416.158} C_VEL
LIN {X 0,Y 119.583,Z 827.641,A -85,B 0,C 180,E1 -30417.548,E2 -30417.548} C_VEL
LIN {X 0,Y 130.05,Z 820.099,A -85,B 0,C 180,E1 -30418.661,E2 -30418.661} C_VEL
LIN {X 0,Y 140.562,Z 811.531,A -85,B 0,C 180,E1 -30419.511,E2 -30419.511} C_VEL
LIN {X 0,Y 151.102,Z 801.751,A -85,B 0,C 180,E1 -30420.377,E2 -30420.377} C_VEL
LIN {X 0,Y 161.667,Z 790.536,A -85,B 0,C 180,E1 -30421.049,E2 -30421.049} C_VEL
LIN {X 0,Y 169.603,Z 780.994,A -85,B 0,C 180,E1 -30421.486,E2 -30421.486} C_VEL
LIN {X 0,Y 177.546,Z 770.195,A -85,B 0,C 180,E1 -30421.853,E2 -30421.853} C_VEL
LIN {X 0,Y 185.319,Z 758.081,A -85,B 0,C 180,E1 -30422.216,E2 -30422.216} C_VEL
LIN {X 0,Y 191.688,Z 746.624,A -85,B 0,C 180,E1 -30422.477,E2 -30422.477} C_VEL
LIN {X 0,Y 197.877,Z 733.609,A -85,B 0,C 180,E1 -30422.697,E2 -30422.697} C_VEL
LIN {X 0,Y 202.739,Z 721.437,A -85,B 0,C 180,E1 -30422.842,E2 -30422.842} C_VEL
LIN {X 0,Y 207.051,Z 708.334,A -85,B 0,C 180,E1 -30422.975,E2 -30422.975} C_VEL
LIN {X 0,Y 210.625,Z 694.501,A -85,B 0,C 180,E1 -30423.102,E2 -30423.102} C_VEL
LIN {X 0,Y 212.044,Z 688.072,A -85,B 0,C 180,E1 -30423.221,E2 -30423.221} C_VEL
LIN {X 0,Y 212.127,Z 690.643,A -85,B 0,C 180,E1 -30425.615,E2 -30425.615} C_VEL
LIN {X 0,Y 212.231,Z 693.397,A -85,B 0,C 180,E1 -30427.4,E2 -30427.4} C_VEL
LIN {X 0,Y 212.37,Z 699.837,A -85,B 0,C 180,E1 -30430.321,E2 -30430.321} C_VEL
LIN {X 0,Y 213.244,Z 710.724,A -85,B 0,C 180,E1 -30435.287,E2 -30435.287} C_VEL
LIN {X 0,Y 215.315,Z 720.217,A -85,B 0,C 180,E1 -30440.042,E2 -30440.042} C_VEL
LIN {X 0,Y 218.686,Z 728.888,A -85,B 0,C 180,E1 -30444.694,E2 -30444.694} C_VEL
LIN {X 0,Y 219.25,Z 729.971,A -85,B 0,C 180,E1 -30445.317,E2 -30445.317} C_VEL
LIN {X 0,Y 220.255,Z 732.871,A -85,B 0,C 180,E1 -30446.633,E2 -30446.633} C_VEL
LIN {X 0,Y 221.939,Z 744.931,A -85,B 0,C 180,E1 -30450.686,E2 -30450.686} C_VEL
LIN {X 0,Y 223.211,Z 747.668,A -85,B 0,C 180,E1 -30451.99,E2 -30451.99} C_VEL
LIN {X 0,Y 237.483,Z 761.727,A -85,B 0,C 180,E1 -30460.621,E2 -30460.621} C_VEL
LIN {X 0,Y 251.088,Z 772.326,A -85,B 0,C 180,E1 -30466.697,E2 -30466.697} C_VEL
LIN {X 0,Y 262.127,Z 780.772,A -85,B 0,C 180,E1 -30471.034,E2 -30471.034} C_VEL
LIN {X 0,Y 269.314,Z 786.352,A -85,B 0,C 180,E1 -30473.995,E2 -30473.995} C_VEL
LIN {X 0,Y 274.65,Z 790.301,A -85,B 0,C 180,E1 -30476.266,E2 -30476.266} C_VEL
LIN {X 0,Y 279.763,Z 794.297,A -85,B 0,C 180,E1 -30478.662,E2 -30478.662} C_VEL
LIN {X 0,Y 285.342,Z 798.361,A -85,B 0,C 180,E1 -30481.387,E2 -30481.387} C_VEL
LIN {X 0,Y 289.889,Z 801.706,A -85,B 0,C 180,E1 -30483.768,E2 -30483.768} C_VEL
LIN {X 0,Y 293.844,Z 804.616,A -85,B 0,C 180,E1 -30486.009,E2 -30486.009} C_VEL
LIN {X 0,Y 299.34,Z 808.275,A -85,B 0,C 180,E1 -30489.38,E2 -30489.38} C_VEL
LIN {X 0,Y 302.911,Z 810.928,A -85,B 0,C 180,E1 -30492.036,E2 -30492.036} C_VEL
LIN {X 0,Y 306.036,Z 813.295,A -85,B 0,C 180,E1 -30494.688,E2 -30494.688} C_VEL
LIN {X 0,Y 309.204,Z 815.381,A -85,B 0,C 180,E1 -30497.782,E2 -30497.782} C_VEL
LIN {X 0,Y 310.94,Z 816.24,A -85,B 0,C 180,E1 -30499.583,E2 -30499.583} C_VEL
LIN {X 0,Y 313.07,Z 817.204,A -85,B 0,C 180,E1 -30502.259,E2 -30502.259} C_VEL
LIN {X 0,Y 314.428,Z 817.965,A -85,B 0,C 180,E1 -30504.871,E2 -30504.871} C_VEL
LIN {X 0,Y 315.378,Z 818.273,A -85,B 0,C 180,E1 -30507.446,E2 -30507.446} C_VEL
LIN {X 0,Y 315.617,Z 818.363,A -85,B 0,C 180,E1 -30508.724,E2 -30508.724} C_VEL
LIN {X 0,Y 315.531,Z 818.398,A -85,B 0,C 180,E1 -30511.276,E2 -30511.276} C_VEL
LIN {X 0,Y 314.909,Z 818.202,A -85,B 0,C 180,E1 -30513.839,E2 -30513.839} C_VEL
LIN {X 0,Y 313.858,Z 817.638,A -85,B 0,C 180,E1 -30516.428,E2 -30516.428} C_VEL
LIN {X 0,Y 312.056,Z 816.792,A -85,B 0,C 180,E1 -30519.07,E2 -30519.07} C_VEL
LIN {X 0,Y 309.235,Z 815.353,A -85,B 0,C 180,E1 -30522.245,E2 -30522.245} C_VEL
LIN {X 0,Y 306.028,Z 813.333,A -85,B 0,C 180,E1 -30525.307,E2 -30525.307} C_VEL
LIN {X 0,Y 302.911,Z 810.962,A -85,B 0,C 180,E1 -30527.964,E2 -30527.964} C_VEL
LIN {X 0,Y 299.345,Z 808.302,A -85,B 0,C 180,E1 -30530.619,E2 -30530.619} C_VEL
LIN {X 0,Y 293.807,Z 804.62,A -85,B 0,C 180,E1 -30533.994,E2 -30533.994} C_VEL
LIN {X 0,Y 288.269,Z 800.479,A -85,B 0,C 180,E1 -30537.146,E2 -30537.146} C_VEL
LIN {X 0,Y 283.062,Z 796.723,A -85,B 0,C 180,E1 -30539.773,E2 -30539.773} C_VEL
LIN {X 0,Y 278.399,Z 793.216,A -85,B 0,C 180,E1 -30542.014,E2 -30542.014} C_VEL
LIN {X 0,Y 272.827,Z 788.956,A -85,B 0,C 180,E1 -30544.521,E2 -30544.521} C_VEL
LIN {X 0,Y 265.745,Z 783.57,A -85,B 0,C 180,E1 -30547.497,E2 -30547.497} C_VEL
LIN {X 0,Y 260.244,Z 779.401,A -85,B 0,C 180,E1 -30549.678,E2 -30549.678} C_VEL
LIN {X 0,Y 253.209,Z 773.845,A -85,B 0,C 180,E1 -30552.478,E2 -30552.478} C_VEL
LIN {X 0,Y 239.522,Z 763.409,A -85,B 0,C 180,E1 -30558.369,E2 -30558.369} C_VEL
LIN {X 0,Y 224.777,Z 749.612,A -85,B 0,C 180,E1 -30566.828,E2 -30566.828} C_VEL
LIN {X 0,Y 216.627,Z 737.697,A -85,B 0,C 180,E1 -30574.026,E2 -30574.026} C_VEL
LIN {X 0,Y 213.105,Z 729.514,A -85,B 0,C 180,E1 -30578.73,E2 -30578.73} C_VEL
LIN {X 0,Y 210.957,Z 720.486,A -85,B 0,C 180,E1 -30583.551,E2 -30583.551} C_VEL
LIN {X 0,Y 210.136,Z 709.017,A -85,B 0,C 180,E1 -30589.096,E2 -30589.096} C_VEL
LIN {X 0,Y 210.489,Z 699.717,A -85,B 0,C 180,E1 -30593.34,E2 -30593.34} C_VEL
LIN {X 0,Y 210.48,Z 697.272,A -85,B 0,C 180,E1 -30594.951,E2 -30594.951} C_VEL
LIN {X 0,Y 205.398,Z 715.158,A -85,B 0,C 180,E1 -30595.107,E2 -30595.107} C_VEL
LIN {X 0,Y 199.669,Z 730.333,A -85,B 0,C 180,E1 -30595.224,E2 -30595.224} C_VEL
LIN {X 0,Y 193.9,Z 742.939,A -85,B 0,C 180,E1 -30595.362,E2 -30595.362} C_VEL
LIN {X 0,Y 187.421,Z 755.025,A -85,B 0,C 180,E1 -30595.537,E2 -30595.537} C_VEL
LIN {X 0,Y 179.664,Z 767.422,A -85,B 0,C 180,E1 -30595.805,E2 -30595.805} C_VEL
LIN {X 0,Y 171.714,Z 778.504,A -85,B 0,C 180,E1 -30596.039,E2 -30596.039} C_VEL
LIN {X 0,Y 162.839,Z 789.325,A -85,B 0,C 180,E1 -30596.405,E2 -30596.405} C_VEL
LIN {X 0,Y 153.093,Z 799.77,A -85,B 0,C 180,E1 -30596.807,E2 -30596.807} C_VEL
LIN {X 0,Y 144.125,Z 808.282,A -85,B 0,C 180,E1 -30597.319,E2 -30597.319} C_VEL
LIN {X 0,Y 133.609,Z 817.142,A -85,B 0,C 180,E1 -30598.011,E2 -30598.011} C_VEL
LIN {X 0,Y 123.018,Z 825.018,A -85,B 0,C 180,E1 -30598.723,E2 -30598.723} C_VEL
LIN {X 0,Y 112.447,Z 831.976,A -85,B 0,C 180,E1 -30599.663,E2 -30599.663} C_VEL
LIN {X 0,Y 101.915,Z 838.115,A -85,B 0,C 180,E1 -30600.845,E2 -30600.845} C_VEL
LIN {X 0,Y 87.957,Z 845.062,A -85,B 0,C 180,E1 -30602.854,E2 -30602.854} C_VEL
LIN {X 0,Y 74.748,Z 850.596,A -85,B 0,C 180,E1 -30605.396,E2 -30605.396} C_VEL
LIN {X 0,Y 63.928,Z 854.448,A -85,B 0,C 180,E1 -30608.351,E2 -30608.351} C_VEL
LIN {X 0,Y 50.654,Z 858.32,A -85,B 0,C 180,E1 -30613.787,E2 -30613.787} C_VEL
LIN {X 0,Y 38.118,Z 861.201,A -85,B 0,C 180,E1 -30622.8,E2 -30622.8} C_VEL
LIN {X 0,Y 27.15,Z 863.118,A -85,B 0,C 180,E1 -30639.054,E2 -30639.054} C_VEL
LIN {X 0,Y 23.005,Z 863.815,A -85,B 0,C 180,E1 -30652.339,E2 -30652.339} C_VEL
LIN {X 0,Y 19.881,Z 864.328,A -85,B 0,C 180,E1 -30690,E2 -30690} C_VEL
LIN {X 0,Y 22.999,Z 863.815,A -85,B 0,C 180,E1 -30727.672,E2 -30727.672} C_VEL
LIN {X 0,Y 32.343,Z 862.353,A -85,B 0,C 180,E1 -30750.362,E2 -30750.362} C_VEL
LIN {X 0,Y 44.267,Z 859.937,A -85,B 0,C 180,E1 -30762.282,E2 -30762.282} C_VEL
LIN {X 0,Y 60.564,Z 855.492,A -85,B 0,C 180,E1 -30770.519,E2 -30770.519} C_VEL
LIN {X 0,Y 70.718,Z 852.114,A -85,B 0,C 180,E1 -30773.61,E2 -30773.61} C_VEL
LIN {X 0,Y 84.486,Z 846.606,A -85,B 0,C 180,E1 -30776.568,E2 -30776.568} C_VEL
LIN {X 0,Y 94.923,Z 841.749,A -85,B 0,C 180,E1 -30778.195,E2 -30778.195} C_VEL
LIN {X 0,Y 109.236,Z 833.898,A -85,B 0,C 180,E1 -30779.999,E2 -30779.999} C_VEL
LIN {X 0,Y 119.491,Z 827.431,A -85,B 0,C 180,E1 -30781.004,E2 -30781.004} C_VEL
LIN {X 0,Y 130.08,Z 819.891,A -85,B 0,C 180,E1 -30781.819,E2 -30781.819} C_VEL
LIN {X 0,Y 140.685,Z 811.321,A -85,B 0,C 180,E1 -30782.444,E2 -30782.444} C_VEL
LIN {X 0,Y 151.319,Z 801.544,A -85,B 0,C 180,E1 -30783.092,E2 -30783.092} C_VEL
LIN {X 0,Y 161.07,Z 791.332,A -85,B 0,C 180,E1 -30783.548,E2 -30783.548} C_VEL
LIN {X 0,Y 169.939,Z 780.788,A -85,B 0,C 180,E1 -30783.897,E2 -30783.897} C_VEL
LIN {X 0,Y 177.869,Z 770.063,A -85,B 0,C 180,E1 -30784.152,E2 -30784.152} C_VEL
LIN {X 0,Y 184.846,Z 759.372,A -85,B 0,C 180,E1 -30784.391,E2 -30784.391} C_VEL
LIN {X 0,Y 192.125,Z 746.418,A -85,B 0,C 180,E1 -30784.593,E2 -30784.593} C_VEL
LIN {X 0,Y 197.895,Z 734.433,A -85,B 0,C 180,E1 -30784.738,E2 -30784.738} C_VEL
LIN {X 0,Y 203.215,Z 721.235,A -85,B 0,C 180,E1 -30784.842,E2 -30784.842} C_VEL
LIN {X 0,Y 207.591,Z 707.97,A -85,B 0,C 180,E1 -30784.945,E2 -30784.945} C_VEL
LIN {X 0,Y 210.486,Z 697.231,A -85,B 0,C 180,E1 -30785.04,E2 -30785.04} C_VEL
LIN {X 0,Y 210.487,Z 699.647,A -85,B 0,C 180,E1 -30786.613,E2 -30786.613} C_VEL
LIN {X 0,Y 210.156,Z 706.042,A -85,B 0,C 180,E1 -30789.564,E2 -30789.564} C_VEL
LIN {X 0,Y 210.487,Z 716.529,A -85,B 0,C 180,E1 -30794.473,E2 -30794.473} C_VEL
LIN {X 0,Y 212.125,Z 725.986,A -85,B 0,C 180,E1 -30799.348,E2 -30799.348} C_VEL
LIN {X 0,Y 215.026,Z 734.567,A -85,B 0,C 180,E1 -30804.112,E2 -30804.112} C_VEL
LIN {X 0,Y 223.211,Z 747.668,A -85,B 0,C 180,E1 -30811.99,E2 -30811.99} C_VEL
LIN {X 0,Y 224.604,Z 750.331,A -85,B 0,C 180,E1 -30813.293,E2 -30813.293} C_VEL
LIN {X 0,Y 227.538,Z 761.424,A -85,B 0,C 180,E1 -30817.389,E2 -30817.389} C_VEL
LIN {X 0,Y 229.228,Z 763.924,A -85,B 0,C 180,E1 -30818.66,E2 -30818.66} C_VEL
LIN {X 0,Y 242.002,Z 774.289,A -85,B 0,C 180,E1 -30825.039,E2 -30825.039} C_VEL
LIN {X 0,Y 251.391,Z 781.362,A -85,B 0,C 180,E1 -30829.009,E2 -30829.009} C_VEL
LIN {X 0,Y 260.069,Z 787.973,A -85,B 0,C 180,E1 -30832.484,E2 -30832.484} C_VEL
LIN {X 0,Y 266.013,Z 792.537,A -85,B 0,C 180,E1 -30834.985,E2 -30834.985} C_VEL
LIN {X 0,Y 271.355,Z 796.498,A -85,B 0,C 180,E1 -30837.322,E2 -30837.322} C_VEL
LIN {X 0,Y 276.518,Z 800.519,A -85,B 0,C 180,E1 -30839.784,E2 -30839.784} C_VEL
LIN {X 0,Y 281.692,Z 804.216,A -85,B 0,C 180,E1 -30842.335,E2 -30842.335} C_VEL
LIN {X 0,Y 286.705,Z 807.986,A -85,B 0,C 180,E1 -30845.09,E2 -30845.09} C_VEL
LIN {X 0,Y 290.307,Z 810.523,A -85,B 0,C 180,E1 -30847.211,E2 -30847.211} C_VEL
LIN {X 0,Y 293.403,Z 812.557,A -85,B 0,C 180,E1 -30849.095,E2 -30849.095} C_VEL
LIN {X 0,Y 296.629,Z 814.842,A -85,B 0,C 180,E1 -30851.388,E2 -30851.388} C_VEL
LIN {X 0,Y 299.79,Z 817.287,A -85,B 0,C 180,E1 -30853.977,E2 -30853.977} C_VEL
LIN {X 0,Y 302.96,Z 819.477,A -85,B 0,C 180,E1 -30856.981,E2 -30856.981} C_VEL
LIN {X 0,Y 305.337,Z 820.757,A -85,B 0,C 180,E1 -30859.389,E2 -30859.389} C_VEL
LIN {X 0,Y 307.571,Z 821.769,A -85,B 0,C 180,E1 -30862.12,E2 -30862.12} C_VEL
LIN {X 0,Y 308.962,Z 822.539,A -85,B 0,C 180,E1 -30864.78,E2 -30864.78} C_VEL
LIN {X 0,Y 309.957,Z 822.889,A -85,B 0,C 180,E1 -30867.401,E2 -30867.401} C_VEL
LIN {X 0,Y 310.217,Z 822.979,A -85,B 0,C 180,E1 -30868.702,E2 -30868.702} C_VEL
LIN {X 0,Y 310.147,Z 822.996,A -85,B 0,C 180,E1 -30871.298,E2 -30871.298} C_VEL
LIN {X 0,Y 309.479,Z 822.785,A -85,B 0,C 180,E1 -30873.906,E2 -30873.906} C_VEL
LIN {X 0,Y 308.372,Z 822.195,A -85,B 0,C 180,E1 -30876.543,E2 -30876.543} C_VEL
LIN {X 0,Y 307.562,Z 821.816,A -85,B 0,C 180,E1 -30877.88,E2 -30877.88} C_VEL
LIN {X 0,Y 305.33,Z 820.75,A -85,B 0,C 180,E1 -30880.611,E2 -30880.611} C_VEL
LIN {X 0,Y 302.544,Z 819.211,A -85,B 0,C 180,E1 -30883.432,E2 -30883.432} C_VEL
LIN {X 0,Y 299.365,Z 817.005,A -85,B 0,C 180,E1 -30886.362,E2 -30886.362} C_VEL
LIN {X 0,Y 295.542,Z 814.025,A -85,B 0,C 180,E1 -30889.446,E2 -30889.446} C_VEL
LIN {X 0,Y 293.123,Z 812.397,A -85,B 0,C 180,E1 -30891.078,E2 -30891.078} C_VEL
LIN {X 0,Y 290.025,Z 810.344,A -85,B 0,C 180,E1 -30892.954,E2 -30892.954} C_VEL
LIN {X 0,Y 285.049,Z 806.724,A -85,B 0,C 180,E1 -30895.855,E2 -30895.855} C_VEL
LIN {X 0,Y 280.109,Z 803.04,A -85,B 0,C 180,E1 -30898.47,E2 -30898.47} C_VEL
LIN {X 0,Y 275.588,Z 799.816,A -85,B 0,C 180,E1 -30900.665,E2 -30900.665} C_VEL
LIN {X 0,Y 269.631,Z 795.118,A -85,B 0,C 180,E1 -30903.48,E2 -30903.48} C_VEL
LIN {X 0,Y 264.116,Z 791.094,A -85,B 0,C 180,E1 -30905.831,E2 -30905.831} C_VEL
LIN {X 0,Y 258.786,Z 786.958,A -85,B 0,C 180,E1 -30908.042,E2 -30908.042} C_VEL
LIN {X 0,Y 247.795,Z 778.521,A -85,B 0,C 180,E1 -30912.489,E2 -30912.489} C_VEL
LIN {X 0,Y 234.169,Z 768.191,A -85,B 0,C 180,E1 -30918.68,E2 -30918.68} C_VEL
LIN {X 0,Y 220.316,Z 754.988,A -85,B 0,C 180,E1 -30927.161,E2 -30927.161} C_VEL
LIN {X 0,Y 213.405,Z 744.812,A -85,B 0,C 180,E1 -30933.603,E2 -30933.603} C_VEL
LIN {X 0,Y 209.601,Z 735.165,A -85,B 0,C 180,E1 -30939.388,E2 -30939.388} C_VEL
LIN {X 0,Y 207.95,Z 726.257,A -85,B 0,C 180,E1 -30944.314,E2 -30944.314} C_VEL
LIN {X 0,Y 207.791,Z 714.216,A -85,B 0,C 180,E1 -30950.264,E2 -30950.264} C_VEL
LIN {X 0,Y 208.256,Z 708.053,A -85,B 0,C 180,E1 -30953.074,E2 -30953.074} C_VEL
LIN {X 0,Y 203.89,Z 721.18,A -85,B 0,C 180,E1 -30953.153,E2 -30953.153} C_VEL
LIN {X 0,Y 197.718,Z 736.281,A -85,B 0,C 180,E1 -30953.231,E2 -30953.231} C_VEL
LIN {X 0,Y 189.091,Z 753.172,A -85,B 0,C 180,E1 -30953.35,E2 -30953.35} C_VEL
LIN {X 0,Y 181.392,Z 765.657,A -85,B 0,C 180,E1 -30953.517,E2 -30953.517} C_VEL
LIN {X 0,Y 172.35,Z 778.299,A -85,B 0,C 180,E1 -30953.682,E2 -30953.682} C_VEL
LIN {X 0,Y 163.443,Z 789.117,A -85,B 0,C 180,E1 -30953.905,E2 -30953.905} C_VEL
LIN {X 0,Y 155.435,Z 797.791,A -85,B 0,C 180,E1 -30954.103,E2 -30954.103} C_VEL
LIN {X 0,Y 145.291,Z 807.5,A -85,B 0,C 180,E1 -30954.449,E2 -30954.449} C_VEL
LIN {X 0,Y 134.049,Z 816.934,A -85,B 0,C 180,E1 -30954.949,E2 -30954.949} C_VEL
LIN {X 0,Y 123.388,Z 824.808,A -85,B 0,C 180,E1 -30955.379,E2 -30955.379} C_VEL
LIN {X 0,Y 112.719,Z 831.766,A -85,B 0,C 180,E1 -30956.008,E2 -30956.008} C_VEL
LIN {X 0,Y 102.065,Z 837.904,A -85,B 0,C 180,E1 -30956.777,E2 -30956.777} C_VEL
LIN {X 0,Y 87.894,Z 844.85,A -85,B 0,C 180,E1 -30958.147,E2 -30958.147} C_VEL
LIN {X 0,Y 77.31,Z 849.326,A -85,B 0,C 180,E1 -30959.438,E2 -30959.438} C_VEL
LIN {X 0,Y 63.284,Z 854.238,A -85,B 0,C 180,E1 -30961.873,E2 -30961.873} C_VEL
LIN {X 0,Y 49.432,Z 858.107,A -85,B 0,C 180,E1 -30965.611,E2 -30965.611} C_VEL
LIN {X 0,Y 35.942,Z 860.989,A -85,B 0,C 180,E1 -30972.136,E2 -30972.136} C_VEL
LIN {X 0,Y 23.307,Z 862.906,A -85,B 0,C 180,E1 -30985.231,E2 -30985.231} C_VEL
LIN {X 0,Y 17.873,Z 863.603,A -85,B 0,C 180,E1 -30998.148,E2 -30998.148} C_VEL
LIN {X 0,Y 12.753,Z 864.117,A -85,B 0,C 180,E1 -31050,E2 -31050} C_VEL
LIN {X 0,Y 17.869,Z 863.603,A -85,B 0,C 180,E1 -31101.867,E2 -31101.867} C_VEL
LIN {X 0,Y 29.453,Z 862.14,A -85,B 0,C 180,E1 -31122.64,E2 -31122.64} C_VEL
LIN {X 0,Y 42.629,Z 859.724,A -85,B 0,C 180,E1 -31131.554,E2 -31131.554} C_VEL
LIN {X 0,Y 59.8,Z 855.281,A -85,B 0,C 180,E1 -31137.359,E2 -31137.359} C_VEL
LIN {X 0,Y 70.281,Z 851.903,A -85,B 0,C 180,E1 -31139.478,E2 -31139.478} C_VEL
LIN {X 0,Y 84.361,Z 846.395,A -85,B 0,C 180,E1 -31141.452,E2 -31141.452} C_VEL
LIN {X 0,Y 94.971,Z 841.538,A -85,B 0,C 180,E1 -31142.561,E2 -31142.561} C_VEL
LIN {X 0,Y 110.03,Z 833.358,A -85,B 0,C 180,E1 -31143.804,E2 -31143.804} C_VEL
LIN {X 0,Y 121.612,Z 826.014,A -85,B 0,C 180,E1 -31144.544,E2 -31144.544} C_VEL
LIN {X 0,Y 132.279,Z 818.308,A -85,B 0,C 180,E1 -31145.018,E2 -31145.018} C_VEL
LIN {X 0,Y 142.485,Z 809.965,A -85,B 0,C 180,E1 -31145.448,E2 -31145.448} C_VEL
LIN {X 0,Y 151.876,Z 801.336,A -85,B 0,C 180,E1 -31145.801,E2 -31145.801} C_VEL
LIN {X 0,Y 161.669,Z 791.125,A -85,B 0,C 180,E1 -31146.073,E2 -31146.073} C_VEL
LIN {X 0,Y 170.573,Z 780.582,A -85,B 0,C 180,E1 -31146.288,E2 -31146.288} C_VEL
LIN {X 0,Y 179.196,Z 768.875,A -85,B 0,C 180,E1 -31146.445,E2 -31146.445} C_VEL
LIN {X 0,Y 186.327,Z 757.819,A -85,B 0,C 180,E1 -31146.593,E2 -31146.593} C_VEL
LIN {X 0,Y 192.825,Z 746.213,A -85,B 0,C 180,E1 -31146.698,E2 -31146.698} C_VEL
LIN {X 0,Y 198.601,Z 734.244,A -85,B 0,C 180,E1 -31146.777,E2 -31146.777} C_VEL
LIN {X 0,Y 203.886,Z 721.175,A -85,B 0,C 180,E1 -31146.832,E2 -31146.832} C_VEL
LIN {X 0,Y 208.257,Z 708.027,A -85,B 0,C 180,E1 -31146.91,E2 -31146.91} C_VEL
LIN {X 0,Y 207.574,Z 720.431,A -85,B 0,C 180,E1 -31152.713,E2 -31152.713} C_VEL
LIN {X 0,Y 208.391,Z 729.979,A -85,B 0,C 180,E1 -31157.669,E2 -31157.669} C_VEL
LIN {X 0,Y 211.227,Z 740.169,A -85,B 0,C 180,E1 -31163.532,E2 -31163.532} C_VEL
LIN {X 0,Y 217.068,Z 750.724,A -85,B 0,C 180,E1 -31170.121,E2 -31170.121} C_VEL
LIN {X 0,Y 228.146,Z 762.951,A -85,B 0,C 180,E1 -31178.031,E2 -31178.031} C_VEL
LIN {X 0,Y 229.228,Z 763.924,A -85,B 0,C 180,E1 -31178.66,E2 -31178.66} C_VEL
LIN {X 0,Y 231.085,Z 766.381,A -85,B 0,C 180,E1 -31179.918,E2 -31179.918} C_VEL
LIN {X 0,Y 234.987,Z 776.88,A -85,B 0,C 180,E1 -31183.951,E2 -31183.951} C_VEL
LIN {X 0,Y 236.998,Z 779.302,A -85,B 0,C 180,E1 -31185.168,E2 -31185.168} C_VEL
LIN {X 0,Y 246.109,Z 786.037,A -85,B 0,C 180,E1 -31189.176,E2 -31189.176} C_VEL
LIN {X 0,Y 255.368,Z 793.031,A -85,B 0,C 180,E1 -31192.949,E2 -31192.949} C_VEL
LIN {X 0,Y 262.662,Z 798.534,A -85,B 0,C 180,E1 -31196.042,E2 -31196.042} C_VEL
LIN {X 0,Y 267.694,Z 802.376,A -85,B 0,C 180,E1 -31198.327,E2 -31198.327} C_VEL
LIN {X 0,Y 272.52,Z 806.045,A -85,B 0,C 180,E1 -31200.661,E2 -31200.661} C_VEL
LIN {X 0,Y 276.871,Z 809.154,A -85,B 0,C 180,E1 -31202.813,E2 -31202.813} C_VEL
LIN {X 0,Y 280.428,Z 811.828,A -85,B 0,C 180,E1 -31204.784,E2 -31204.784} C_VEL
LIN {X 0,Y 284.723,Z 814.865,A -85,B 0,C 180,E1 -31207.293,E2 -31207.293} C_VEL
LIN {X 0,Y 289.166,Z 817.856,A -85,B 0,C 180,E1 -31210.108,E2 -31210.108} C_VEL
LIN {X 0,Y 291.402,Z 819.468,A -85,B 0,C 180,E1 -31211.728,E2 -31211.728} C_VEL
LIN {X 0,Y 293.394,Z 821.073,A -85,B 0,C 180,E1 -31213.366,E2 -31213.366} C_VEL
LIN {X 0,Y 296.591,Z 823.348,A -85,B 0,C 180,E1 -31216.293,E2 -31216.293} C_VEL
LIN {X 0,Y 299.498,Z 825.013,A -85,B 0,C 180,E1 -31219.18,E2 -31219.18} C_VEL
LIN {X 0,Y 301.809,Z 826.049,A -85,B 0,C 180,E1 -31221.969,E2 -31221.969} C_VEL
LIN {X 0,Y 303.315,Z 826.849,A -85,B 0,C 180,E1 -31224.682,E2 -31224.682} C_VEL
LIN {X 0,Y 304.346,Z 827.254,A -85,B 0,C 180,E1 -31227.353,E2 -31227.353} C_VEL
LIN {X 0,Y 304.629,Z 827.348,A -85,B 0,C 180,E1 -31228.678,E2 -31228.678} C_VEL
LIN {X 0,Y 304.556,Z 827.362,A -85,B 0,C 180,E1 -31231.322,E2 -31231.322} C_VEL
LIN {X 0,Y 303.849,Z 827.124,A -85,B 0,C 180,E1 -31233.979,E2 -31233.979} C_VEL
LIN {X 0,Y 302.656,Z 826.504,A -85,B 0,C 180,E1 -31236.667,E2 -31236.667} C_VEL
LIN {X 0,Y 300.727,Z 825.624,A -85,B 0,C 180,E1 -31239.415,E2 -31239.415} C_VEL
LIN {X 0,Y 298.095,Z 824.243,A -85,B 0,C 180,E1 -31242.25,E2 -31242.25} C_VEL
LIN {X 0,Y 295.001,Z 822.248,A -85,B 0,C 180,E1 -31245.192,E2 -31245.192} C_VEL
LIN {X 0,Y 293.278,Z 821.006,A -85,B 0,C 180,E1 -31246.712,E2 -31246.712} C_VEL
LIN {X 0,Y 290.2,Z 818.549,A -85,B 0,C 180,E1 -31249.182,E2 -31249.182} C_VEL
LIN {X 0,Y 286.556,Z 816.155,A -85,B 0,C 180,E1 -31251.585,E2 -31251.585} C_VEL
LIN {X 0,Y 282.448,Z 813.36,A -85,B 0,C 180,E1 -31254.039,E2 -31254.039} C_VEL
LIN {X 0,Y 278.407,Z 810.304,A -85,B 0,C 180,E1 -31256.347,E2 -31256.347} C_VEL
LIN {X 0,Y 275.39,Z 808.064,A -85,B 0,C 180,E1 -31257.959,E2 -31257.959} C_VEL
LIN {X 0,Y 269.737,Z 803.962,A -85,B 0,C 180,E1 -31260.705,E2 -31260.705} C_VEL
LIN {X 0,Y 264.497,Z 799.845,A -85,B 0,C 180,E1 -31263.177,E2 -31263.177} C_VEL
LIN {X 0,Y 259.029,Z 795.848,A -85,B 0,C 180,E1 -31265.516,E2 -31265.516} C_VEL
LIN {X 0,Y 251.629,Z 790.18,A -85,B 0,C 180,E1 -31268.553,E2 -31268.553} C_VEL
LIN {X 0,Y 242.329,Z 783.149,A -85,B 0,C 180,E1 -31272.475,E2 -31272.475} C_VEL
LIN {X 0,Y 229.139,Z 773.203,A -85,B 0,C 180,E1 -31278.744,E2 -31278.744} C_VEL
LIN {X 0,Y 214.798,Z 759.094,A -85,B 0,C 180,E1 -31288.285,E2 -31288.285} C_VEL
LIN {X 0,Y 207.961,Z 747.211,A -85,B 0,C 180,E1 -31296.076,E2 -31296.076} C_VEL
LIN {X 0,Y 205.31,Z 737.373,A -85,B 0,C 180,E1 -31302.057,E2 -31302.057} C_VEL
LIN {X 0,Y 204.856,Z 724.773,A -85,B 0,C 180,E1 -31308.859,E2 -31308.859} C_VEL
LIN {X 0,Y 205.214,Z 720.128,A -85,B 0,C 180,E1 -31311.086,E2 -31311.086} C_VEL
LIN {X 0,Y 204.854,Z 720.993,A -85,B 0,C 180,E1 -31311.177,E2 -31311.177} C_VEL
LIN {X 0,Y 198.682,Z 736.08,A -85,B 0,C 180,E1 -31311.194,E2 -31311.194} C_VEL
LIN {X 0,Y 190.226,Z 752.669,A -85,B 0,C 180,E1 -31311.216,E2 -31311.216} C_VEL
LIN {X 0,Y 181.896,Z 766.092,A -85,B 0,C 180,E1 -31311.293,E2 -31311.293} C_VEL
LIN {X 0,Y 173.277,Z 778.094,A -85,B 0,C 180,E1 -31311.345,E2 -31311.345} C_VEL
LIN {X 0,Y 164.358,Z 788.909,A -85,B 0,C 180,E1 -31311.421,E2 -31311.421} C_VEL
LIN {X 0,Y 154.55,Z 799.356,A -85,B 0,C 180,E1 -31311.507,E2 -31311.507} C_VEL
LIN {X 0,Y 145.304,Z 808.042,A -85,B 0,C 180,E1 -31311.657,E2 -31311.657} C_VEL
LIN {X 0,Y 134.871,Z 816.725,A -85,B 0,C 180,E1 -31311.909,E2 -31311.909} C_VEL
LIN {X 0,Y 124.176,Z 824.599,A -85,B 0,C 180,E1 -31312.067,E2 -31312.067} C_VEL
LIN {X 0,Y 113.447,Z 831.557,A -85,B 0,C 180,E1 -31312.38,E2 -31312.38} C_VEL
LIN {X 0,Y 102.725,Z 837.694,A -85,B 0,C 180,E1 -31312.748,E2 -31312.748} C_VEL
LIN {X 0,Y 88.423,Z 844.638,A -85,B 0,C 180,E1 -31313.463,E2 -31313.463} C_VEL
LIN {X 0,Y 77.715,Z 849.116,A -85,B 0,C 180,E1 -31314.122,E2 -31314.122} C_VEL
LIN {X 0,Y 63.462,Z 854.027,A -85,B 0,C 180,E1 -31315.322,E2 -31315.322} C_VEL
LIN {X 0,Y 49.253,Z 857.896,A -85,B 0,C 180,E1 -31317.227,E2 -31317.227} C_VEL
LIN {X 0,Y 35.141,Z 860.778,A -85,B 0,C 180,E1 -31320.564,E2 -31320.564} C_VEL
LIN {X 0,Y 21.264,Z 862.697,A -85,B 0,C 180,E1 -31327.475,E2 -31327.475} C_VEL
LIN {X 0,Y 14.575,Z 863.391,A -85,B 0,C 180,E1 -31335.335,E2 -31335.335} C_VEL
LIN {X 0,Y 5.64,Z 863.907,A -85,B 0,C 180,E1 -31410,E2 -31410} C_VEL
LIN {X 0,Y 14.573,Z 863.391,A -85,B 0,C 180,E1 -31484.685,E2 -31484.685} C_VEL
LIN {X 0,Y 28.156,Z 861.93,A -85,B 0,C 180,E1 -31496.779,E2 -31496.779} C_VEL
LIN {X 0,Y 42.178,Z 859.512,A -85,B 0,C 180,E1 -31501.331,E2 -31501.331} C_VEL
LIN {X 0,Y 59.902,Z 855.071,A -85,B 0,C 180,E1 -31504.264,E2 -31504.264} C_VEL
LIN {X 0,Y 72.742,Z 850.914,A -85,B 0,C 180,E1 -31505.543,E2 -31505.543} C_VEL
LIN {X 0,Y 84.851,Z 846.184,A -85,B 0,C 180,E1 -31506.331,E2 -31506.331} C_VEL
LIN {X 0,Y 95.566,Z 841.328,A -85,B 0,C 180,E1 -31506.888,E2 -31506.888} C_VEL
LIN {X 0,Y 110.258,Z 833.432,A -85,B 0,C 180,E1 -31507.508,E2 -31507.508} C_VEL
LIN {X 0,Y 120.606,Z 827.012,A -85,B 0,C 180,E1 -31507.86,E2 -31507.86} C_VEL
LIN {X 0,Y 131.319,Z 819.475,A -85,B 0,C 180,E1 -31508.081,E2 -31508.081} C_VEL
LIN {X 0,Y 142.037,Z 810.9,A -85,B 0,C 180,E1 -31508.279,E2 -31508.279} C_VEL
LIN {X 0,Y 152.769,Z 801.128,A -85,B 0,C 180,E1 -31508.48,E2 -31508.48} C_VEL
LIN {X 0,Y 163.478,Z 789.911,A -85,B 0,C 180,E1 -31508.599,E2 -31508.599} C_VEL
LIN {X 0,Y 171.507,Z 780.375,A -85,B 0,C 180,E1 -31508.672,E2 -31508.672} C_VEL
LIN {X 0,Y 179.903,Z 769.008,A -85,B 0,C 180,E1 -31508.698,E2 -31508.698} C_VEL
LIN {X 0,Y 186.657,Z 758.662,A -85,B 0,C 180,E1 -31508.758,E2 -31508.758} C_VEL
LIN {X 0,Y 193.786,Z 746.006,A -85,B 0,C 180,E1 -31508.794,E2 -31508.794} C_VEL
LIN {X 0,Y 199.627,Z 733.899,A -85,B 0,C 180,E1 -31508.805,E2 -31508.805} C_VEL
LIN {X 0,Y 204.844,Z 720.988,A -85,B 0,C 180,E1 -31508.8,E2 -31508.8} C_VEL
LIN {X 0,Y 205.195,Z 720.181,A -85,B 0,C 180,E1 -31508.915,E2 -31508.915} C_VEL
LIN {X 0,Y 204.71,Z 730.027,A -85,B 0,C 180,E1 -31513.905,E2 -31513.905} C_VEL
LIN {X 0,Y 205.626,Z 739.049,A -85,B 0,C 180,E1 -31518.947,E2 -31518.947} C_VEL
LIN {X 0,Y 207.962,Z 747.209,A -85,B 0,C 180,E1 -31523.924,E2 -31523.924} C_VEL
LIN {X 0,Y 214.821,Z 759.093,A -85,B 0,C 180,E1 -31531.725,E2 -31531.725} C_VEL
LIN {X 0,Y 229.141,Z 773.196,A -85,B 0,C 180,E1 -31541.255,E2 -31541.255} C_VEL
LIN {X 0,Y 236.998,Z 779.302,A -85,B 0,C 180,E1 -31545.168,E2 -31545.168} C_VEL
LIN {X 0,Y 239.126,Z 781.72,A -85,B 0,C 180,E1 -31546.366,E2 -31546.366} C_VEL
LIN {X 0,Y 243.446,Z 791.854,A -85,B 0,C 180,E1 -31550.303,E2 -31550.303} C_VEL
LIN {X 0,Y 245.672,Z 794.228,A -85,B 0,C 180,E1 -31551.461,E2 -31551.461} C_VEL
LIN {X 0,Y 253.695,Z 800.311,A -85,B 0,C 180,E1 -31554.806,E2 -31554.806} C_VEL
LIN {X 0,Y 259.218,Z 804.431,A -85,B 0,C 180,E1 -31557.19,E2 -31557.19} C_VEL
LIN {X 0,Y 264.529,Z 808.518,A -85,B 0,C 180,E1 -31559.683,E2 -31559.683} C_VEL
LIN {X 0,Y 269.873,Z 812.411,A -85,B 0,C 180,E1 -31562.302,E2 -31562.302} C_VEL
LIN {X 0,Y 274.588,Z 815.852,A -85,B 0,C 180,E1 -31564.828,E2 -31564.828} C_VEL
LIN {X 0,Y 280.177,Z 819.845,A -85,B 0,C 180,E1 -31568.141,E2 -31568.141} C_VEL
LIN {X 0,Y 283.604,Z 822.099,A -85,B 0,C 180,E1 -31570.333,E2 -31570.333} C_VEL
LIN {X 0,Y 286.952,Z 824.648,A -85,B 0,C 180,E1 -31572.909,E2 -31572.909} C_VEL
LIN {X 0,Y 290.403,Z 827.159,A -85,B 0,C 180,E1 -31575.995,E2 -31575.995} C_VEL
LIN {X 0,Y 293.499,Z 829.002,A -85,B 0,C 180,E1 -31579.039,E2 -31579.039} C_VEL
LIN {X 0,Y 295.837,Z 830.067,A -85,B 0,C 180,E1 -31581.805,E2 -31581.805} C_VEL
LIN {X 0,Y 297.449,Z 830.922,A -85,B 0,C 180,E1 -31584.577,E2 -31584.577} C_VEL
LIN {X 0,Y 298.549,Z 831.367,A -85,B 0,C 180,E1 -31587.302,E2 -31587.302} C_VEL
LIN {X 0,Y 298.842,Z 831.475,A -85,B 0,C 180,E1 -31588.652,E2 -31588.652} C_VEL
LIN {X 0,Y 298.77,Z 831.485,A -85,B 0,C 180,E1 -31591.348,E2 -31591.348} C_VEL
LIN {X 0,Y 298.534,Z 831.351,A -85,B 0,C 180,E1 -31592.699,E2 -31592.699} C_VEL
LIN {X 0,Y 297.488,Z 830.909,A -85,B 0,C 180,E1 -31595.422,E2 -31595.422} C_VEL
LIN {X 0,Y 295.832,Z 830.109,A -85,B 0,C 180,E1 -31598.195,E2 -31598.195} C_VEL
LIN {X 0,Y 293.423,Z 828.964,A -85,B 0,C 180,E1 -31601.047,E2 -31601.047} C_VEL
LIN {X 0,Y 290.1,Z 826.955,A -85,B 0,C 180,E1 -31604.296,E2 -31604.296} C_VEL
LIN {X 0,Y 286.859,Z 824.617,A -85,B 0,C 180,E1 -31607.161,E2 -31607.161} C_VEL
LIN {X 0,Y 283.587,Z 822.107,A -85,B 0,C 180,E1 -31609.657,E2 -31609.657} C_VEL
LIN {X 0,Y 279.674,Z 819.539,A -85,B 0,C 180,E1 -31612.144,E2 -31612.144} C_VEL
LIN {X 0,Y 274.541,Z 815.851,A -85,B 0,C 180,E1 -31615.174,E2 -31615.174} C_VEL
LIN {X 0,Y 269.221,Z 811.921,A -85,B 0,C 180,E1 -31618.026,E2 -31618.026} C_VEL
LIN {X 0,Y 262.771,Z 807.151,A -85,B 0,C 180,E1 -31621.146,E2 -31621.146} C_VEL
LIN {X 0,Y 257.144,Z 802.844,A -85,B 0,C 180,E1 -31623.72,E2 -31623.72} C_VEL
LIN {X 0,Y 249.754,Z 797.263,A -85,B 0,C 180,E1 -31626.835,E2 -31626.835} C_VEL
LIN {X 0,Y 239.049,Z 789.27,A -85,B 0,C 180,E1 -31631.437,E2 -31631.437} C_VEL
LIN {X 0,Y 225.558,Z 779.346,A -85,B 0,C 180,E1 -31637.941,E2 -31637.941} C_VEL
LIN {X 0,Y 212.109,Z 766.765,A -85,B 0,C 180,E1 -31646.859,E2 -31646.859} C_VEL
LIN {X 0,Y 205.022,Z 755.655,A -85,B 0,C 180,E1 -31654.629,E2 -31654.629} C_VEL
LIN {X 0,Y 202.168,Z 746.277,A -85,B 0,C 180,E1 -31660.717,E2 -31660.717} C_VEL
LIN {X 0,Y 201.526,Z 736.571,A -85,B 0,C 180,E1 -31666.437,E2 -31666.437} C_VEL
LIN {X 0,Y 201.77,Z 731.753,A -85,B 0,C 180,E1 -31669.058,E2 -31669.058} C_VEL
LIN {X 0,Y 201.221,Z 732.825,A -85,B 0,C 180,E1 -31669.186,E2 -31669.186} C_VEL
LIN {X 0,Y 195.004,Z 745.8,A -85,B 0,C 180,E1 -31669.135,E2 -31669.135} C_VEL
LIN {X 0,Y 186.986,Z 759.956,A -85,B 0,C 180,E1 -31669.083,E2 -31669.083} C_VEL
LIN {X 0,Y 176.273,Z 775.605,A -85,B 0,C 180,E1 -31669.045,E2 -31669.045} C_VEL
LIN {X 0,Y 167.362,Z 786.69,A -85,B 0,C 180,E1 -31668.98,E2 -31668.98} C_VEL
LIN {X 0,Y 157.547,Z 797.377,A -85,B 0,C 180,E1 -31668.923,E2 -31668.923} C_VEL
LIN {X 0,Y 147.038,Z 807.375,A -85,B 0,C 180,E1 -31668.889,E2 -31668.889} C_VEL
LIN {X 0,Y 136.069,Z 816.517,A -85,B 0,C 180,E1 -31668.912,E2 -31668.912} C_VEL
LIN {X 0,Y 125.368,Z 824.39,A -85,B 0,C 180,E1 -31668.816,E2 -31668.816} C_VEL
LIN {X 0,Y 114.63,Z 831.346,A -85,B 0,C 180,E1 -31668.796,E2 -31668.796} C_VEL
LIN {X 0,Y 103.882,Z 837.484,A -85,B 0,C 180,E1 -31668.8,E2 -31668.8} C_VEL
LIN {X 0,Y 89.531,Z 844.427,A -85,B 0,C 180,E1 -31668.873,E2 -31668.873} C_VEL
LIN {X 0,Y 74.844,Z 850.323,A -85,B 0,C 180,E1 -31668.886,E2 -31668.886} C_VEL
LIN {X 0,Y 64.456,Z 853.816,A -85,B 0,C 180,E1 -31668.9,E2 -31668.9} C_VEL
LIN {X 0,Y 50.127,Z 857.683,A -85,B 0,C 180,E1 -31668.931,E2 -31668.931} C_VEL
LIN {X 0,Y 35.8,Z 860.568,A -85,B 0,C 180,E1 -31668.971,E2 -31668.971} C_VEL
LIN {X 0,Y 21.544,Z 862.487,A -85,B 0,C 180,E1 -31668.135,E2 -31668.135} C_VEL
LIN {X 0,Y 14.444,Z 863.177,A -85,B 0,C 180,E1 -31666.678,E2 -31666.678} C_VEL
LIN {X 0,Y 1.493,Z 863.696,A -85,B 0,C 180,E1 -31590,E2 -31590} C_VEL
LIN {X 0,Y 14.445,Z 863.177,A -85,B 0,C 180,E1 -31513.341,E2 -31513.341} C_VEL
LIN {X 0,Y 28.667,Z 861.72,A -85,B 0,C 180,E1 -31511.3,E2 -31511.3} C_VEL
LIN {X 0,Y 42.955,Z 859.3,A -85,B 0,C 180,E1 -31510.992,E2 -31510.992} C_VEL
LIN {X 0,Y 60.871,Z 854.86,A -85,B 0,C 180,E1 -31511.081,E2 -31511.081} C_VEL
LIN {X 0,Y 72.87,Z 851.033,A -85,B 0,C 180,E1 -31511.12,E2 -31511.12} C_VEL
LIN {X 0,Y 85.944,Z 845.973,A -85,B 0,C 180,E1 -31511.109,E2 -31511.109} C_VEL
LIN {X 0,Y 96.695,Z 841.119,A -85,B 0,C 180,E1 -31511.131,E2 -31511.131} C_VEL
LIN {X 0,Y 110.683,Z 833.661,A -85,B 0,C 180,E1 -31511.186,E2 -31511.186} C_VEL
LIN {X 0,Y 121.794,Z 826.803,A -85,B 0,C 180,E1 -31511.204,E2 -31511.204} C_VEL
LIN {X 0,Y 132.512,Z 819.268,A -85,B 0,C 180,E1 -31511.142,E2 -31511.142} C_VEL
LIN {X 0,Y 143.247,Z 810.691,A -85,B 0,C 180,E1 -31511.123,E2 -31511.123} C_VEL
LIN {X 0,Y 153.985,Z 800.922,A -85,B 0,C 180,E1 -31511.112,E2 -31511.112} C_VEL
LIN {X 0,Y 164.701,Z 789.702,A -85,B 0,C 180,E1 -31511.062,E2 -31511.062} C_VEL
LIN {X 0,Y 173.608,Z 779.029,A -85,B 0,C 180,E1 -31510.989,E2 -31510.989} C_VEL
LIN {X 0,Y 181.538,Z 768.188,A -85,B 0,C 180,E1 -31510.925,E2 -31510.925} C_VEL
LIN {X 0,Y 188.77,Z 756.959,A -85,B 0,C 180,E1 -31510.908,E2 -31510.908} C_VEL
LIN {X 0,Y 195.894,Z 744.06,A -85,B 0,C 180,E1 -31510.857,E2 -31510.857} C_VEL
LIN {X 0,Y 201.224,Z 732.806,A -85,B 0,C 180,E1 -31510.805,E2 -31510.805} C_VEL
LIN {X 0,Y 201.764,Z 731.915,A -85,B 0,C 180,E1 -31511.043,E2 -31511.043} C_VEL
LIN {X 0,Y 201.535,Z 741.235,A -85,B 0,C 180,E1 -31516.199,E2 -31516.199} C_VEL
LIN {X 0,Y 203.313,Z 751.158,A -85,B 0,C 180,E1 -31522.348,E2 -31522.348} C_VEL
LIN {X 0,Y 209.059,Z 762.744,A -85,B 0,C 180,E1 -31530.281,E2 -31530.281} C_VEL
LIN {X 0,Y 219.694,Z 774.42,A -85,B 0,C 180,E1 -31538.613,E2 -31538.613} C_VEL
LIN {X 0,Y 232.031,Z 784.291,A -85,B 0,C 180,E1 -31545.38,E2 -31545.38} C_VEL
LIN {X 0,Y 240.777,Z 790.628,A -85,B 0,C 180,E1 -31549.367,E2 -31549.367} C_VEL
LIN {X 0,Y 245.672,Z 794.228,A -85,B 0,C 180,E1 -31551.461,E2 -31551.461} C_VEL
LIN {X 0,Y 247.851,Z 796.647,A -85,B 0,C 180,E1 -31552.606,E2 -31552.606} C_VEL
LIN {X 0,Y 249.896,Z 801.613,A -85,B 0,C 180,E1 -31554.529,E2 -31554.529} C_VEL
LIN {X 0,Y 251.349,Z 805.552,A -85,B 0,C 180,E1 -31556.086,E2 -31556.086} C_VEL
LIN {X 0,Y 253.07,Z 808.066,A -85,B 0,C 180,E1 -31557.254,E2 -31557.254} C_VEL
LIN {X 0,Y 253.854,Z 808.695,A -85,B 0,C 180,E1 -31557.637,E2 -31557.637} C_VEL
LIN {X 0,Y 259.232,Z 812.845,A -85,B 0,C 180,E1 -31560.173,E2 -31560.173} C_VEL
LIN {X 0,Y 262.864,Z 815.501,A -85,B 0,C 180,E1 -31561.919,E2 -31561.919} C_VEL
LIN {X 0,Y 268.17,Z 819.351,A -85,B 0,C 180,E1 -31564.703,E2 -31564.703} C_VEL
LIN {X 0,Y 273.36,Z 823.119,A -85,B 0,C 180,E1 -31567.749,E2 -31567.749} C_VEL
LIN {X 0,Y 278.166,Z 826.315,A -85,B 0,C 180,E1 -31570.826,E2 -31570.826} C_VEL
LIN {X 0,Y 280.332,Z 827.973,A -85,B 0,C 180,E1 -31572.492,E2 -31572.492} C_VEL
LIN {X 0,Y 283.975,Z 830.672,A -85,B 0,C 180,E1 -31575.672,E2 -31575.672} C_VEL
LIN {X 0,Y 286.875,Z 832.485,A -85,B 0,C 180,E1 -31578.501,E2 -31578.501} C_VEL
LIN {X 0,Y 289.673,Z 833.807,A -85,B 0,C 180,E1 -31581.63,E2 -31581.63} C_VEL
LIN {X 0,Y 291.414,Z 834.724,A -85,B 0,C 180,E1 -31584.464,E2 -31584.464} C_VEL
LIN {X 0,Y 292.561,Z 835.214,A -85,B 0,C 180,E1 -31587.246,E2 -31587.246} C_VEL
LIN {X 0,Y 292.881,Z 835.308,A -85,B 0,C 180,E1 -31588.625,E2 -31588.625} C_VEL
LIN {X 0,Y 292.804,Z 835.321,A -85,B 0,C 180,E1 -31591.375,E2 -31591.375} C_VEL
LIN {X 0,Y 292.547,Z 835.195,A -85,B 0,C 180,E1 -31592.754,E2 -31592.754} C_VEL
LIN {X 0,Y 291.436,Z 834.719,A -85,B 0,C 180,E1 -31595.535,E2 -31595.535} C_VEL
LIN {X 0,Y 289.669,Z 833.842,A -85,B 0,C 180,E1 -31598.37,E2 -31598.37} C_VEL
LIN {X 0,Y 286.891,Z 832.486,A -85,B 0,C 180,E1 -31601.515,E2 -31601.515} C_VEL
LIN {X 0,Y 283.995,Z 830.68,A -85,B 0,C 180,E1 -31604.327,E2 -31604.327} C_VEL
LIN {X 0,Y 280.206,Z 827.884,A -85,B 0,C 180,E1 -31607.62,E2 -31607.62} C_VEL
LIN {X 0,Y 276.834,Z 825.434,A -85,B 0,C 180,E1 -31610.065,E2 -31610.065} C_VEL
LIN {X 0,Y 272.478,Z 822.526,A -85,B 0,C 180,E1 -31612.761,E2 -31612.761} C_VEL
LIN {X 0,Y 268.123,Z 819.352,A -85,B 0,C 180,E1 -31615.3,E2 -31615.3} C_VEL
LIN {X 0,Y 262.86,Z 815.488,A -85,B 0,C 180,E1 -31618.079,E2 -31618.079} C_VEL
LIN {X 0,Y 255.651,Z 810.109,A -85,B 0,C 180,E1 -31621.549,E2 -31621.549} C_VEL
LIN {X 0,Y 249.458,Z 805.424,A -85,B 0,C 180,E1 -31624.295,E2 -31624.295} C_VEL
LIN {X 0,Y 240.788,Z 798.997,A -85,B 0,C 180,E1 -31627.996,E2 -31627.996} C_VEL
LIN {X 0,Y 232.747,Z 793.16,A -85,B 0,C 180,E1 -31631.628,E2 -31631.628} C_VEL
LIN {X 0,Y 219.236,Z 783.302,A -85,B 0,C 180,E1 -31638.565,E2 -31638.565} C_VEL
LIN {X 0,Y 205.67,Z 769.838,A -85,B 0,C 180,E1 -31648.678,E2 -31648.678} C_VEL
LIN {X 0,Y 199.637,Z 757.974,A -85,B 0,C 180,E1 -31657.218,E2 -31657.218} C_VEL
LIN {X 0,Y 198.044,Z 748.417,A -85,B 0,C 180,E1 -31663.508,E2 -31663.508} C_VEL
LIN {X 0,Y 198.071,Z 742.971,A -85,B 0,C 180,E1 -31666.771,E2 -31666.771} C_VEL
LIN {X 0,Y 197.357,Z 743.856,A -85,B 0,C 180,E1 -31667.113,E2 -31667.113} C_VEL
LIN {X 0,Y 190.246,Z 756.755,A -85,B 0,C 180,E1 -31666.985,E2 -31666.985} C_VEL
LIN {X 0,Y 182.804,Z 768.295,A -85,B 0,C 180,E1 -31666.886,E2 -31666.886} C_VEL
LIN {X 0,Y 174.221,Z 779.966,A -85,B 0,C 180,E1 -31666.698,E2 -31666.698} C_VEL
LIN {X 0,Y 164.418,Z 791.508,A -85,B 0,C 180,E1 -31666.511,E2 -31666.511} C_VEL
LIN {X 0,Y 151.952,Z 804.192,A -85,B 0,C 180,E1 -31666.229,E2 -31666.229} C_VEL
LIN {X 0,Y 139.417,Z 814.931,A -85,B 0,C 180,E1 -31666.017,E2 -31666.017} C_VEL
LIN {X 0,Y 126.957,Z 824.181,A -85,B 0,C 180,E1 -31665.633,E2 -31665.633} C_VEL
LIN {X 0,Y 116.245,Z 831.136,A -85,B 0,C 180,E1 -31665.309,E2 -31665.309} C_VEL
LIN {X 0,Y 105.521,Z 837.274,A -85,B 0,C 180,E1 -31664.955,E2 -31664.955} C_VEL
LIN {X 0,Y 91.203,Z 844.215,A -85,B 0,C 180,E1 -31664.412,E2 -31664.412} C_VEL
LIN {X 0,Y 76.562,Z 850.113,A -85,B 0,C 180,E1 -31663.584,E2 -31663.584} C_VEL
LIN {X 0,Y 62.662,Z 854.65,A -85,B 0,C 180,E1 -31662.424,E2 -31662.424} C_VEL
LIN {X 0,Y 44.91,Z 859.087,A -85,B 0,C 180,E1 -31659.872,E2 -31659.872} C_VEL
LIN {X 0,Y 30.892,Z 861.51,A -85,B 0,C 180,E1 -31655.505,E2 -31655.505} C_VEL
LIN {X 0,Y 17.553,Z 862.963,A -85,B 0,C 180,E1 -31643.204,E2 -31643.204} C_VEL
LIN {X 0,Y 8.636,Z 863.485,A -85,B 0,C 180,E1 -31590,E2 -31590} C_VEL
LIN {X 0,Y 17.555,Z 862.963,A -85,B 0,C 180,E1 -31536.807,E2 -31536.807} C_VEL
LIN {X 0,Y 30.892,Z 861.51,A -85,B 0,C 180,E1 -31524.496,E2 -31524.496} C_VEL
LIN {X 0,Y 44.897,Z 859.088,A -85,B 0,C 180,E1 -31520.085,E2 -31520.085} C_VEL
LIN {X 0,Y 62.664,Z 854.649,A -85,B 0,C 180,E1 -31517.583,E2 -31517.583} C_VEL
LIN {X 0,Y 76.564,Z 850.112,A -85,B 0,C 180,E1 -31516.422,E2 -31516.422} C_VEL
LIN {X 0,Y 91.199,Z 844.216,A -85,B 0,C 180,E1 -31515.581,E2 -31515.581} C_VEL
LIN {X 0,Y 105.504,Z 837.276,A -85,B 0,C 180,E1 -31515.011,E2 -31515.011} C_VEL
LIN {X 0,Y 121.612,Z 827.801,A -85,B 0,C 180,E1 -31514.541,E2 -31514.541} C_VEL
LIN {X 0,Y 134.077,Z 819.06,A -85,B 0,C 180,E1 -31514.14,E2 -31514.14} C_VEL
LIN {X 0,Y 144.803,Z 810.482,A -85,B 0,C 180,E1 -31513.91,E2 -31513.91} C_VEL
LIN {X 0,Y 155.526,Z 800.714,A -85,B 0,C 180,E1 -31513.705,E2 -31513.705} C_VEL
LIN {X 0,Y 166.219,Z 789.495,A -85,B 0,C 180,E1 -31513.479,E2 -31513.479} C_VEL
LIN {X 0,Y 175.106,Z 778.824,A -85,B 0,C 180,E1 -31513.278,E2 -31513.278} C_VEL
LIN {X 0,Y 183.583,Z 767.167,A -85,B 0,C 180,E1 -31513.115,E2 -31513.115} C_VEL
LIN {X 0,Y 191.141,Z 755.256,A -85,B 0,C 180,E1 -31513.006,E2 -31513.006} C_VEL
LIN {X 0,Y 197.357,Z 743.856,A -85,B 0,C 180,E1 -31512.887,E2 -31512.887} C_VEL
LIN {X 0,Y 198.058,Z 742.997,A -85,B 0,C 180,E1 -31513.23,E2 -31513.23} C_VEL
LIN {X 0,Y 198.776,Z 754.985,A -85,B 0,C 180,E1 -31520.705,E2 -31520.705} C_VEL
LIN {X 0,Y 203.462,Z 766.564,A -85,B 0,C 180,E1 -31528.919,E2 -31528.919} C_VEL
LIN {X 0,Y 213.557,Z 778.463,A -85,B 0,C 180,E1 -31537.833,E2 -31537.833} C_VEL
LIN {X 0,Y 226.7,Z 788.955,A -85,B 0,C 180,E1 -31545.481,E2 -31545.481} C_VEL
LIN {X 0,Y 235.366,Z 795.11,A -85,B 0,C 180,E1 -31549.589,E2 -31549.589} C_VEL
LIN {X 0,Y 244.503,Z 801.73,A -85,B 0,C 180,E1 -31553.593,E2 -31553.593} C_VEL
LIN {X 0,Y 252.003,Z 807.322,A -85,B 0,C 180,E1 -31556.787,E2 -31556.787} C_VEL
LIN {X 0,Y 253.854,Z 808.695,A -85,B 0,C 180,E1 -31557.637,E2 -31557.637} C_VEL
LIN {X 0,Y 255.259,Z 810.156,A -85,B 0,C 180,E1 -31558.403,E2 -31558.403} C_VEL
LIN {X 0,Y 256.814,Z 813.604,A -85,B 0,C 180,E1 -31559.961,E2 -31559.961} C_VEL
LIN {X 0,Y 258.58,Z 819.683,A -85,B 0,C 180,E1 -31562.73,E2 -31562.73} C_VEL
LIN {X 0,Y 260.257,Z 821.607,A -85,B 0,C 180,E1 -31563.915,E2 -31563.915} C_VEL
LIN {X 0,Y 264.936,Z 825.068,A -85,B 0,C 180,E1 -31566.553,E2 -31566.553} C_VEL
LIN {X 0,Y 269.956,Z 828.494,A -85,B 0,C 180,E1 -31569.588,E2 -31569.588} C_VEL
LIN {X 0,Y 273.451,Z 830.964,A -85,B 0,C 180,E1 -31572.037,E2 -31572.037} C_VEL
LIN {X 0,Y 277.362,Z 833.849,A -85,B 0,C 180,E1 -31575.322,E2 -31575.322} C_VEL
LIN {X 0,Y 280.568,Z 835.908,A -85,B 0,C 180,E1 -31578.44,E2 -31578.44} C_VEL
LIN {X 0,Y 283.297,Z 837.276,A -85,B 0,C 180,E1 -31581.44,E2 -31581.44} C_VEL
LIN {X 0,Y 284.389,Z 837.793,A -85,B 0,C 180,E1 -31582.902,E2 -31582.902} C_VEL
LIN {X 0,Y 285.798,Z 838.558,A -85,B 0,C 180,E1 -31585.769,E2 -31585.769} C_VEL
LIN {X 0,Y 286.364,Z 838.72,A -85,B 0,C 180,E1 -31587.187,E2 -31587.187} C_VEL
LIN {X 0,Y 286.698,Z 838.822,A -85,B 0,C 180,E1 -31588.595,E2 -31588.595} C_VEL
LIN {X 0,Y 286.637,Z 838.823,A -85,B 0,C 180,E1 -31591.405,E2 -31591.405} C_VEL
LIN {X 0,Y 286.357,Z 838.697,A -85,B 0,C 180,E1 -31592.813,E2 -31592.813} C_VEL
LIN {X 0,Y 285.195,Z 838.233,A -85,B 0,C 180,E1 -31595.657,E2 -31595.657} C_VEL
LIN {X 0,Y 283.809,Z 837.534,A -85,B 0,C 180,E1 -31597.898,E2 -31597.898} C_VEL
LIN {X 0,Y 282.022,Z 836.683,A -85,B 0,C 180,E1 -31600.046,E2 -31600.046} C_VEL
LIN {X 0,Y 279.052,Z 835.02,A -85,B 0,C 180,E1 -31603.101,E2 -31603.101} C_VEL
LIN {X 0,Y 276.743,Z 833.44,A -85,B 0,C 180,E1 -31605.201,E2 -31605.201} C_VEL
LIN {X 0,Y 273.421,Z 830.926,A -85,B 0,C 180,E1 -31608.004,E2 -31608.004} C_VEL
LIN {X 0,Y 269.953,Z 828.509,A -85,B 0,C 180,E1 -31610.411,E2 -31610.411} C_VEL
LIN {X 0,Y 264.92,Z 825.1,A -85,B 0,C 180,E1 -31613.448,E2 -31613.448} C_VEL
LIN {X 0,Y 261.415,Z 822.466,A -85,B 0,C 180,E1 -31615.477,E2 -31615.477} C_VEL
LIN {X 0,Y 255.704,Z 818.323,A -85,B 0,C 180,E1 -31618.417,E2 -31618.417} C_VEL
LIN {X 0,Y 248.37,Z 812.757,A -85,B 0,C 180,E1 -31621.909,E2 -31621.909} C_VEL
LIN {X 0,Y 240.818,Z 807.249,A -85,B 0,C 180,E1 -31625.201,E2 -31625.201} C_VEL
LIN {X 0,Y 233.455,Z 801.975,A -85,B 0,C 180,E1 -31628.492,E2 -31628.492} C_VEL
LIN {X 0,Y 224.634,Z 795.833,A -85,B 0,C 180,E1 -31632.674,E2 -31632.674} C_VEL
LIN {X 0,Y 213.456,Z 787.654,A -85,B 0,C 180,E1 -31638.816,E2 -31638.816} C_VEL
LIN {X 0,Y 202.281,Z 776.82,A -85,B 0,C 180,E1 -31647.417,E2 -31647.417} C_VEL
LIN {X 0,Y 196.716,Z 767.517,A -85,B 0,C 180,E1 -31654.614,E2 -31654.614} C_VEL
LIN {X 0,Y 194.445,Z 758.702,A -85,B 0,C 180,E1 -31661.017,E2 -31661.017} C_VEL
LIN {X 0,Y 194.245,Z 753.013,A -85,B 0,C 180,E1 -31664.768,E2 -31664.768} C_VEL
LIN {X 0,Y 193.187,Z 754.508,A -85,B 0,C 180,E1 -31664.946,E2 -31664.946} C_VEL
LIN {X 0,Y 185.71,Z 766.406,A -85,B 0,C 180,E1 -31664.748,E2 -31664.748} C_VEL
LIN {X 0,Y 177.757,Z 777.478,A -85,B 0,C 180,E1 -31664.514,E2 -31664.514} C_VEL
LIN {X 0,Y 169.792,Z 787.279,A -85,B 0,C 180,E1 -31664.225,E2 -31664.225} C_VEL
LIN {X 0,Y 159.139,Z 798.736,A -85,B 0,C 180,E1 -31663.845,E2 -31663.845} C_VEL
LIN {X 0,Y 150.247,Z 807.148,A -85,B 0,C 180,E1 -31663.51,E2 -31663.51} C_VEL
LIN {X 0,Y 139.544,Z 816.1,A -85,B 0,C 180,E1 -31663.116,E2 -31663.116} C_VEL
LIN {X 0,Y 128.93,Z 823.971,A -85,B 0,C 180,E1 -31662.536,E2 -31662.536} C_VEL
LIN {X 0,Y 116.496,Z 831.978,A -85,B 0,C 180,E1 -31661.832,E2 -31661.832} C_VEL
LIN {X 0,Y 104.068,Z 838.88,A -85,B 0,C 180,E1 -31660.986,E2 -31660.986} C_VEL
LIN {X 0,Y 93.407,Z 844.003,A -85,B 0,C 180,E1 -31660.133,E2 -31660.133} C_VEL
LIN {X 0,Y 79.264,Z 849.773,A -85,B 0,C 180,E1 -31658.586,E2 -31658.586} C_VEL
LIN {X 0,Y 65.205,Z 854.439,A -85,B 0,C 180,E1 -31656.367,E2 -31656.367} C_VEL
LIN {X 0,Y 47.874,Z 858.875,A -85,B 0,C 180,E1 -31651.738,E2 -31651.738} C_VEL
LIN {X 0,Y 34.5,Z 861.299,A -85,B 0,C 180,E1 -31644.569,E2 -31644.569} C_VEL
LIN {X 0,Y 22.601,Z 862.75,A -85,B 0,C 180,E1 -31628.455,E2 -31628.455} C_VEL
LIN {X 0,Y 15.766,Z 863.274,A -85,B 0,C 180,E1 -31590,E2 -31590} C_VEL
LIN {X 0,Y 22.604,Z 862.749,A -85,B 0,C 180,E1 -31551.551,E2 -31551.551} C_VEL
LIN {X 0,Y 34.501,Z 861.299,A -85,B 0,C 180,E1 -31535.432,E2 -31535.432} C_VEL
LIN {X 0,Y 47.862,Z 858.875,A -85,B 0,C 180,E1 -31528.235,E2 -31528.235} C_VEL
LIN {X 0,Y 65.209,Z 854.439,A -85,B 0,C 180,E1 -31523.64,E2 -31523.64} C_VEL
LIN {X 0,Y 79.266,Z 849.773,A -85,B 0,C 180,E1 -31521.417,E2 -31521.417} C_VEL
LIN {X 0,Y 93.402,Z 844.004,A -85,B 0,C 180,E1 -31519.859,E2 -31519.859} C_VEL
LIN {X 0,Y 110.464,Z 835.537,A -85,B 0,C 180,E1 -31518.548,E2 -31518.548} C_VEL
LIN {X 0,Y 125.394,Z 826.384,A -85,B 0,C 180,E1 -31517.677,E2 -31517.677} C_VEL
LIN {X 0,Y 136,Z 818.853,A -85,B 0,C 180,E1 -31517.062,E2 -31517.062} C_VEL
LIN {X 0,Y 148.296,Z 808.866,A -85,B 0,C 180,E1 -31516.572,E2 -31516.572} C_VEL
LIN {X 0,Y 157.375,Z 800.507,A -85,B 0,C 180,E1 -31516.236,E2 -31516.236} C_VEL
LIN {X 0,Y 168.037,Z 789.286,A -85,B 0,C 180,E1 -31515.861,E2 -31515.861} C_VEL
LIN {X 0,Y 176.879,Z 778.619,A -85,B 0,C 180,E1 -31515.526,E2 -31515.526} C_VEL
LIN {X 0,Y 185.587,Z 766.594,A -85,B 0,C 180,E1 -31515.263,E2 -31515.263} C_VEL
LIN {X 0,Y 193.185,Z 754.511,A -85,B 0,C 180,E1 -31515.054,E2 -31515.054} C_VEL
LIN {X 0,Y 194.242,Z 753.016,A -85,B 0,C 180,E1 -31515.23,E2 -31515.23} C_VEL
LIN {X 0,Y 194.941,Z 761.808,A -85,B 0,C 180,E1 -31521.132,E2 -31521.132} C_VEL
LIN {X 0,Y 199.541,Z 772.97,A -85,B 0,C 180,E1 -31529.543,E2 -31529.543} C_VEL
LIN {X 0,Y 209.666,Z 784.449,A -85,B 0,C 180,E1 -31538.663,E2 -31538.663} C_VEL
LIN {X 0,Y 221.426,Z 793.62,A -85,B 0,C 180,E1 -31545.713,E2 -31545.713} C_VEL
LIN {X 0,Y 230.594,Z 799.99,A -85,B 0,C 180,E1 -31550.207,E2 -31550.207} C_VEL
LIN {X 0,Y 238.938,Z 805.832,A -85,B 0,C 180,E1 -31553.967,E2 -31553.967} C_VEL
LIN {X 0,Y 246.295,Z 811.21,A -85,B 0,C 180,E1 -31557.17,E2 -31557.17} C_VEL
LIN {X 0,Y 252.115,Z 815.667,A -85,B 0,C 180,E1 -31559.884,E2 -31559.884} C_VEL
LIN {X 0,Y 257.21,Z 819.394,A -85,B 0,C 180,E1 -31562.322,E2 -31562.322} C_VEL
LIN {X 0,Y 260.257,Z 821.607,A -85,B 0,C 180,E1 -31563.915,E2 -31563.915} C_VEL
LIN {X 0,Y 261.842,Z 823.514,A -85,B 0,C 180,E1 -31565.09,E2 -31565.09} C_VEL
LIN {X 0,Y 262.72,Z 827.267,A -85,B 0,C 180,E1 -31567.082,E2 -31567.082} C_VEL
LIN {X 0,Y 263.122,Z 830.184,A -85,B 0,C 180,E1 -31568.709,E2 -31568.709} C_VEL
LIN {X 0,Y 264.017,Z 831.969,A -85,B 0,C 180,E1 -31569.937,E2 -31569.937} C_VEL
LIN {X 0,Y 264.525,Z 832.392,A -85,B 0,C 180,E1 -31570.344,E2 -31570.344} C_VEL
LIN {X 0,Y 266.496,Z 833.752,A -85,B 0,C 180,E1 -31571.691,E2 -31571.691} C_VEL
LIN {X 0,Y 270.486,Z 836.713,A -85,B 0,C 180,E1 -31574.94,E2 -31574.94} C_VEL
LIN {X 0,Y 273.841,Z 838.923,A -85,B 0,C 180,E1 -31578.152,E2 -31578.152} C_VEL
LIN {X 0,Y 276.751,Z 840.442,A -85,B 0,C 180,E1 -31581.236,E2 -31581.236} C_VEL
LIN {X 0,Y 277.92,Z 840.957,A -85,B 0,C 180,E1 -31582.736,E2 -31582.736} C_VEL
LIN {X 0,Y 279.407,Z 841.755,A -85,B 0,C 180,E1 -31585.672,E2 -31585.672} C_VEL
LIN {X 0,Y 280.01,Z 841.944,A -85,B 0,C 180,E1 -31587.123,E2 -31587.123} C_VEL
LIN {X 0,Y 280.382,Z 842.051,A -85,B 0,C 180,E1 -31588.564,E2 -31588.564} C_VEL
LIN {X 0,Y 280.327,Z 842.048,A -85,B 0,C 180,E1 -31591.437,E2 -31591.437} C_VEL
LIN {X 0,Y 280.008,Z 841.919,A -85,B 0,C 180,E1 -31592.877,E2 -31592.877} C_VEL
LIN {X 0,Y 278.767,Z 841.399,A -85,B 0,C 180,E1 -31595.788,E2 -31595.788} C_VEL
LIN {X 0,Y 277.068,Z 840.607,A -85,B 0,C 180,E1 -31598.41,E2 -31598.41} C_VEL
LIN {X 0,Y 273.897,Z 838.927,A -85,B 0,C 180,E1 -31601.845,E2 -31601.845} C_VEL
LIN {X 0,Y 270.481,Z 836.731,A -85,B 0,C 180,E1 -31605.06,E2 -31605.06} C_VEL
LIN {X 0,Y 266.509,Z 833.74,A -85,B 0,C 180,E1 -31608.317,E2 -31608.317} C_VEL
LIN {X 0,Y 262.945,Z 831.329,A -85,B 0,C 180,E1 -31610.696,E2 -31610.696} C_VEL
LIN {X 0,Y 259.342,Z 828.873,A -85,B 0,C 180,E1 -31612.873,E2 -31612.873} C_VEL
LIN {X 0,Y 255.77,Z 826.219,A -85,B 0,C 180,E1 -31614.939,E2 -31614.939} C_VEL
LIN {X 0,Y 252.128,Z 823.558,A -85,B 0,C 180,E1 -31616.877,E2 -31616.877} C_VEL
LIN {X 0,Y 247.101,Z 819.916,A -85,B 0,C 180,E1 -31619.339,E2 -31619.339} C_VEL
LIN {X 0,Y 240.922,Z 815.182,A -85,B 0,C 180,E1 -31622.226,E2 -31622.226} C_VEL
LIN {X 0,Y 231.543,Z 808.586,A -85,B 0,C 180,E1 -31626.453,E2 -31626.453} C_VEL
LIN {X 0,Y 220.809,Z 801.321,A -85,B 0,C 180,E1 -31631.588,E2 -31631.588} C_VEL
LIN {X 0,Y 209.5,Z 793.385,A -85,B 0,C 180,E1 -31637.862,E2 -31637.862} C_VEL
LIN {X 0,Y 196.175,Z 780.359,A -85,B 0,C 180,E1 -31648.824,E2 -31648.824} C_VEL
LIN {X 0,Y 191.19,Z 769.808,A -85,B 0,C 180,E1 -31657.295,E2 -31657.295} C_VEL
LIN {X 0,Y 190.242,Z 763.15,A -85,B 0,C 180,E1 -31662.256,E2 -31662.256} C_VEL
LIN {X 0,Y 188.867,Z 764.513,A -85,B 0,C 180,E1 -31662.682,E2 -31662.682} C_VEL
LIN {X 0,Y 179.794,Z 777.273,A -85,B 0,C 180,E1 -31662.321,E2 -31662.321} C_VEL
LIN {X 0,Y 171.876,Z 787.071,A -85,B 0,C 180,E1 -31661.928,E2 -31661.928} C_VEL
LIN {X 0,Y 161.281,Z 798.528,A -85,B 0,C 180,E1 -31661.398,E2 -31661.398} C_VEL
LIN {X 0,Y 150.671,Z 808.5,A -85,B 0,C 180,E1 -31660.827,E2 -31660.827} C_VEL
LIN {X 0,Y 140.032,Z 817.268,A -85,B 0,C 180,E1 -31660.222,E2 -31660.222} C_VEL
LIN {X 0,Y 127.745,Z 826.176,A -85,B 0,C 180,E1 -31659.269,E2 -31659.269} C_VEL
LIN {X 0,Y 113.663,Z 834.923,A -85,B 0,C 180,E1 -31658.042,E2 -31658.042} C_VEL
LIN {X 0,Y 99.593,Z 842.24,A -85,B 0,C 180,E1 -31656.541,E2 -31656.541} C_VEL
LIN {X 0,Y 85.637,Z 848.274,A -85,B 0,C 180,E1 -31654.517,E2 -31654.517} C_VEL
LIN {X 0,Y 71.836,Z 853.185,A -85,B 0,C 180,E1 -31651.701,E2 -31651.701} C_VEL
LIN {X 0,Y 58.308,Z 857.047,A -85,B 0,C 180,E1 -31647.534,E2 -31647.534} C_VEL
LIN {X 0,Y 45.261,Z 859.935,A -85,B 0,C 180,E1 -31640.929,E2 -31640.929} C_VEL
LIN {X 0,Y 33.454,Z 861.86,A -85,B 0,C 180,E1 -31629.067,E2 -31629.067} C_VEL
LIN {X 0,Y 24.805,Z 862.838,A -85,B 0,C 180,E1 -31606.459,E2 -31606.459} C_VEL
LIN {X 0,Y 22.888,Z 863.064,A -85,B 0,C 180,E1 -31590,E2 -31590} C_VEL
LIN {X 0,Y 28.582,Z 862.536,A -85,B 0,C 180,E1 -31560.543,E2 -31560.543} C_VEL
LIN {X 0,Y 39.127,Z 861.087,A -85,B 0,C 180,E1 -31544.073,E2 -31544.073} C_VEL
LIN {X 0,Y 51.672,Z 858.663,A -85,B 0,C 180,E1 -31535.309,E2 -31535.309} C_VEL
LIN {X 0,Y 68.426,Z 854.229,A -85,B 0,C 180,E1 -31529.19,E2 -31529.19} C_VEL
LIN {X 0,Y 82.179,Z 849.562,A -85,B 0,C 180,E1 -31526.111,E2 -31526.111} C_VEL
LIN {X 0,Y 96.091,Z 843.792,A -85,B 0,C 180,E1 -31523.905,E2 -31523.905} C_VEL
LIN {X 0,Y 112.076,Z 835.811,A -85,B 0,C 180,E1 -31522.1,E2 -31522.1} C_VEL
LIN {X 0,Y 125.997,Z 827.378,A -85,B 0,C 180,E1 -31520.888,E2 -31520.888} C_VEL
LIN {X 0,Y 138.274,Z 818.645,A -85,B 0,C 180,E1 -31519.903,E2 -31519.903} C_VEL
LIN {X 0,Y 148.917,Z 810.063,A -85,B 0,C 180,E1 -31519.29,E2 -31519.29} C_VEL
LIN {X 0,Y 159.523,Z 800.3,A -85,B 0,C 180,E1 -31518.704,E2 -31518.704} C_VEL
LIN {X 0,Y 170.14,Z 789.077,A -85,B 0,C 180,E1 -31518.187,E2 -31518.187} C_VEL
LIN {X 0,Y 178.925,Z 778.413,A -85,B 0,C 180,E1 -31517.732,E2 -31517.732} C_VEL
LIN {X 0,Y 186.826,Z 767.513,A -85,B 0,C 180,E1 -31517.393,E2 -31517.393} C_VEL
LIN {X 0,Y 188.648,Z 764.852,A -85,B 0,C 180,E1 -31517.339,E2 -31517.339} C_VEL
LIN {X 0,Y 190.226,Z 763.175,A -85,B 0,C 180,E1 -31517.746,E2 -31517.746} C_VEL
LIN {X 0,Y 192.587,Z 774.004,A -85,B 0,C 180,E1 -31525.97,E2 -31525.97} C_VEL
LIN {X 0,Y 199.939,Z 784.956,A -85,B 0,C 180,E1 -31535.049,E2 -31535.049} C_VEL
LIN {X 0,Y 212.573,Z 795.612,A -85,B 0,C 180,E1 -31543.97,E2 -31543.97} C_VEL
LIN {X 0,Y 224.287,Z 803.672,A -85,B 0,C 180,E1 -31550.147,E2 -31550.147} C_VEL
LIN {X 0,Y 233.373,Z 809.861,A -85,B 0,C 180,E1 -31554.399,E2 -31554.399} C_VEL
LIN {X 0,Y 240.914,Z 815.192,A -85,B 0,C 180,E1 -31557.777,E2 -31557.777} C_VEL
LIN {X 0,Y 248.323,Z 820.833,A -85,B 0,C 180,E1 -31561.241,E2 -31561.241} C_VEL
LIN {X 0,Y 253.089,Z 824.254,A -85,B 0,C 180,E1 -31563.622,E2 -31563.622} C_VEL
LIN {X 0,Y 257.072,Z 827.135,A -85,B 0,C 180,E1 -31565.791,E2 -31565.791} C_VEL
LIN {X 0,Y 260.527,Z 829.649,A -85,B 0,C 180,E1 -31567.811,E2 -31567.811} C_VEL
LIN {X 0,Y 264.525,Z 832.392,A -85,B 0,C 180,E1 -31570.344,E2 -31570.344} C_VEL
LIN {X 0,Y 265.577,Z 833.989,A -85,B 0,C 180,E1 -31571.557,E2 -31571.557} C_VEL
LIN {X 0,Y 265.513,Z 837.036,A -85,B 0,C 180,E1 -31573.593,E2 -31573.593} C_VEL
LIN {X 0,Y 265.201,Z 839.373,A -85,B 0,C 180,E1 -31575.251,E2 -31575.251} C_VEL
LIN {X 0,Y 265.631,Z 840.682,A -85,B 0,C 180,E1 -31576.507,E2 -31576.507} C_VEL
LIN {X 0,Y 266.004,Z 840.995,A -85,B 0,C 180,E1 -31576.923,E2 -31576.923} C_VEL
LIN {X 0,Y 268.571,Z 842.531,A -85,B 0,C 180,E1 -31579.445,E2 -31579.445} C_VEL
LIN {X 0,Y 270.21,Z 843.345,A -85,B 0,C 180,E1 -31581.244,E2 -31581.244} C_VEL
LIN {X 0,Y 271.253,Z 843.8,A -85,B 0,C 180,E1 -31582.557,E2 -31582.557} C_VEL
LIN {X 0,Y 272.189,Z 844.275,A -85,B 0,C 180,E1 -31584.072,E2 -31584.072} C_VEL
LIN {X 0,Y 273.502,Z 844.891,A -85,B 0,C 180,E1 -31587.054,E2 -31587.054} C_VEL
LIN {X 0,Y 273.924,Z 845.002,A -85,B 0,C 180,E1 -31588.53,E2 -31588.53} C_VEL
LIN {X 0,Y 273.879,Z 844.995,A -85,B 0,C 180,E1 -31591.47,E2 -31591.47} C_VEL
LIN {X 0,Y 273.501,Z 844.864,A -85,B 0,C 180,E1 -31592.946,E2 -31592.946} C_VEL
LIN {X 0,Y 272.191,Z 844.271,A -85,B 0,C 180,E1 -31595.928,E2 -31595.928} C_VEL
LIN {X 0,Y 271.249,Z 843.806,A -85,B 0,C 180,E1 -31597.443,E2 -31597.443} C_VEL
LIN {X 0,Y 270,Z 843.273,A -85,B 0,C 180,E1 -31598.985,E2 -31598.985} C_VEL
LIN {X 0,Y 267.003,Z 841.603,A -85,B 0,C 180,E1 -31602.156,E2 -31602.156} C_VEL
LIN {X 0,Y 263.407,Z 839.207,A -85,B 0,C 180,E1 -31605.474,E2 -31605.474} C_VEL
LIN {X 0,Y 259.474,Z 836.315,A -85,B 0,C 180,E1 -31608.562,E2 -31608.562} C_VEL
LIN {X 0,Y 255.833,Z 833.858,A -85,B 0,C 180,E1 -31610.933,E2 -31610.933} C_VEL
LIN {X 0,Y 250.368,Z 829.935,A -85,B 0,C 180,E1 -31614.179,E2 -31614.179} C_VEL
LIN {X 0,Y 244.771,Z 825.91,A -85,B 0,C 180,E1 -31617.117,E2 -31617.117} C_VEL
LIN {X 0,Y 238.763,Z 821.424,A -85,B 0,C 180,E1 -31620.025,E2 -31620.025} C_VEL
LIN {X 0,Y 232.39,Z 816.892,A -85,B 0,C 180,E1 -31622.98,E2 -31622.98} C_VEL
LIN {X 0,Y 225.1,Z 811.983,A -85,B 0,C 180,E1 -31626.384,E2 -31626.384} C_VEL
LIN {X 0,Y 215.163,Z 805.486,A -85,B 0,C 180,E1 -31631.301,E2 -31631.301} C_VEL
LIN {X 0,Y 203.962,Z 797.852,A -85,B 0,C 180,E1 -31637.786,E2 -31637.786} C_VEL
LIN {X 0,Y 192.828,Z 787.565,A -85,B 0,C 180,E1 -31646.957,E2 -31646.957} C_VEL
LIN {X 0,Y 186.881,Z 776.33,A -85,B 0,C 180,E1 -31656.669,E2 -31656.669} C_VEL
LIN {X 0,Y 186.101,Z 772.091,A -85,B 0,C 180,E1 -31660.131,E2 -31660.131} C_VEL
LIN {X 0,Y 184.554,Z 773.809,A -85,B 0,C 180,E1 -31660.322,E2 -31660.322} C_VEL
LIN {X 0,Y 174.239,Z 786.862,A -85,B 0,C 180,E1 -31659.682,E2 -31659.682} C_VEL
LIN {X 0,Y 163.702,Z 798.321,A -85,B 0,C 180,E1 -31659.026,E2 -31659.026} C_VEL
LIN {X 0,Y 153.185,Z 808.291,A -85,B 0,C 180,E1 -31658.284,E2 -31658.284} C_VEL
LIN {X 0,Y 142.621,Z 817.06,A -85,B 0,C 180,E1 -31657.507,E2 -31657.507} C_VEL
LIN {X 0,Y 130.461,Z 825.967,A -85,B 0,C 180,E1 -31656.317,E2 -31656.317} C_VEL
LIN {X 0,Y 116.542,Z 834.714,A -85,B 0,C 180,E1 -31654.762,E2 -31654.762} C_VEL
LIN {X 0,Y 102.689,Z 842.026,A -85,B 0,C 180,E1 -31652.835,E2 -31652.835} C_VEL
LIN {X 0,Y 88.987,Z 848.062,A -85,B 0,C 180,E1 -31650.312,E2 -31650.312} C_VEL
LIN {X 0,Y 75.521,Z 852.975,A -85,B 0,C 180,E1 -31646.879,E2 -31646.879} C_VEL
LIN {X 0,Y 62.488,Z 856.835,A -85,B 0,C 180,E1 -31641.931,E2 -31641.931} C_VEL
LIN {X 0,Y 50.129,Z 859.725,A -85,B 0,C 180,E1 -31634.505,E2 -31634.505} C_VEL
LIN {X 0,Y 39.314,Z 861.65,A -85,B 0,C 180,E1 -31622.431,E2 -31622.431} C_VEL
LIN {X 0,Y 31.739,Z 862.628,A -85,B 0,C 180,E1 -31602.793,E2 -31602.793} C_VEL
LIN {X 0,Y 30.038,Z 862.852,A -85,B 0,C 180,E1 -31590,E2 -31590} C_VEL
LIN {X 0,Y 35.01,Z 862.322,A -85,B 0,C 180,E1 -31566.329,E2 -31566.329} C_VEL
LIN {X 0,Y 47.548,Z 860.236,A -85,B 0,C 180,E1 -31547.646,E2 -31547.646} C_VEL
LIN {X 0,Y 56.165,Z 858.45,A -85,B 0,C 180,E1 -31541.343,E2 -31541.343} C_VEL
LIN {X 0,Y 72.23,Z 854.018,A -85,B 0,C 180,E1 -31534.205,E2 -31534.205} C_VEL
LIN {X 0,Y 85.595,Z 849.352,A -85,B 0,C 180,E1 -31530.446,E2 -31530.446} C_VEL
LIN {X 0,Y 99.226,Z 843.581,A -85,B 0,C 180,E1 -31527.707,E2 -31527.707} C_VEL
LIN {X 0,Y 114.044,Z 836.121,A -85,B 0,C 180,E1 -31525.554,E2 -31525.554} C_VEL
LIN {X 0,Y 128.735,Z 827.166,A -85,B 0,C 180,E1 -31523.878,E2 -31523.878} C_VEL
LIN {X 0,Y 140.878,Z 818.436,A -85,B 0,C 180,E1 -31522.648,E2 -31522.648} C_VEL
LIN {X 0,Y 153.188,Z 808.29,A -85,B 0,C 180,E1 -31521.719,E2 -31521.719} C_VEL
LIN {X 0,Y 163.721,Z 798.32,A -85,B 0,C 180,E1 -31520.991,E2 -31520.991} C_VEL
LIN {X 0,Y 174.241,Z 786.86,A -85,B 0,C 180,E1 -31520.32,E2 -31520.32} C_VEL
LIN {X 0,Y 184.564,Z 773.806,A -85,B 0,C 180,E1 -31519.685,E2 -31519.685} C_VEL
LIN {X 0,Y 186.113,Z 772.073,A -85,B 0,C 180,E1 -31519.868,E2 -31519.868} C_VEL
LIN {X 0,Y 189.585,Z 782.79,A -85,B 0,C 180,E1 -31528.81,E2 -31528.81} C_VEL
LIN {X 0,Y 199.809,Z 794.517,A -85,B 0,C 180,E1 -31539.28,E2 -31539.28} C_VEL
LIN {X 0,Y 211.761,Z 803.33,A -85,B 0,C 180,E1 -31546.898,E2 -31546.898} C_VEL
LIN {X 0,Y 220.428,Z 808.961,A -85,B 0,C 180,E1 -31551.364,E2 -31551.364} C_VEL
LIN {X 0,Y 227.743,Z 813.777,A -85,B 0,C 180,E1 -31554.861,E2 -31554.861} C_VEL
LIN {X 0,Y 235.317,Z 818.908,A -85,B 0,C 180,E1 -31558.339,E2 -31558.339} C_VEL
LIN {X 0,Y 243.167,Z 824.736,A -85,B 0,C 180,E1 -31562.086,E2 -31562.086} C_VEL
LIN {X 0,Y 248.731,Z 828.77,A -85,B 0,C 180,E1 -31564.924,E2 -31564.924} C_VEL
LIN {X 0,Y 254.259,Z 832.731,A -85,B 0,C 180,E1 -31568.091,E2 -31568.091} C_VEL
LIN {X 0,Y 258.295,Z 835.501,A -85,B 0,C 180,E1 -31570.618,E2 -31570.618} C_VEL
LIN {X 0,Y 261.259,Z 837.628,A -85,B 0,C 180,E1 -31572.789,E2 -31572.789} C_VEL
LIN {X 0,Y 263.423,Z 839.202,A -85,B 0,C 180,E1 -31574.527,E2 -31574.527} C_VEL
LIN {X 0,Y 266.004,Z 840.995,A -85,B 0,C 180,E1 -31576.923,E2 -31576.923} C_VEL
LIN {X 0,Y 266.659,Z 842.075,A -85,B 0,C 180,E1 -31578.164,E2 -31578.164} C_VEL
LIN {X 0,Y 266.367,Z 843.391,A -85,B 0,C 180,E1 -31579.411,E2 -31579.411} C_VEL
LIN {X 0,Y 265.031,Z 845.864,A -85,B 0,C 180,E1 -31581.932,E2 -31581.932} C_VEL
LIN {X 0,Y 265.036,Z 846.636,A -85,B 0,C 180,E1 -31583.216,E2 -31583.216} C_VEL
LIN {X 0,Y 265.27,Z 846.763,A -85,B 0,C 180,E1 -31583.643,E2 -31583.643} C_VEL
LIN {X 0,Y 266.208,Z 847.284,A -85,B 0,C 180,E1 -31585.457,E2 -31585.457} C_VEL
LIN {X 0,Y 267.202,Z 847.642,A -85,B 0,C 180,E1 -31588.132,E2 -31588.132} C_VEL
LIN {X 0,Y 267.405,Z 847.728,A -85,B 0,C 180,E1 -31590,E2 -31590} C_VEL
LIN {X 0,Y 267.199,Z 847.668,A -85,B 0,C 180,E1 -31591.846,E2 -31591.846} C_VEL
LIN {X 0,Y 266.21,Z 847.265,A -85,B 0,C 180,E1 -31594.543,E2 -31594.543} C_VEL
LIN {X 0,Y 265.473,Z 846.847,A -85,B 0,C 180,E1 -31596.079,E2 -31596.079} C_VEL
LIN {X 0,Y 264.419,Z 846.343,A -85,B 0,C 180,E1 -31597.637,E2 -31597.637} C_VEL
LIN {X 0,Y 261.609,Z 844.965,A -85,B 0,C 180,E1 -31600.839,E2 -31600.839} C_VEL
LIN {X 0,Y 259.524,Z 843.681,A -85,B 0,C 180,E1 -31602.869,E2 -31602.869} C_VEL
LIN {X 0,Y 255.953,Z 841.213,A -85,B 0,C 180,E1 -31606.049,E2 -31606.049} C_VEL
LIN {X 0,Y 252.352,Z 838.595,A -85,B 0,C 180,E1 -31608.758,E2 -31608.758} C_VEL
LIN {X 0,Y 247.805,Z 835.495,A -85,B 0,C 180,E1 -31611.635,E2 -31611.635} C_VEL
LIN {X 0,Y 242.657,Z 831.792,A -85,B 0,C 180,E1 -31614.582,E2 -31614.582} C_VEL
LIN {X 0,Y 237.315,Z 827.915,A -85,B 0,C 180,E1 -31617.324,E2 -31617.324} C_VEL
LIN {X 0,Y 229.662,Z 822.425,A -85,B 0,C 180,E1 -31621.038,E2 -31621.038} C_VEL
LIN {X 0,Y 220.079,Z 816.195,A -85,B 0,C 180,E1 -31625.596,E2 -31625.596} C_VEL
LIN {X 0,Y 209.476,Z 809.569,A -85,B 0,C 180,E1 -31630.986,E2 -31630.986} C_VEL
LIN {X 0,Y 197.264,Z 801.369,A -85,B 0,C 180,E1 -31638.431,E2 -31638.431} C_VEL
LIN {X 0,Y 185.838,Z 789.956,A -85,B 0,C 180,E1 -31649.301,E2 -31649.301} C_VEL
LIN {X 0,Y 181.98,Z 780.745,A -85,B 0,C 180,E1 -31657.64,E2 -31657.64} C_VEL
LIN {X 0,Y 180.283,Z 782.527,A -85,B 0,C 180,E1 -31657.778,E2 -31657.778} C_VEL
LIN {X 0,Y 168.127,Z 796.342,A -85,B 0,C 180,E1 -31656.87,E2 -31656.87} C_VEL
LIN {X 0,Y 157.728,Z 806.517,A -85,B 0,C 180,E1 -31655.981,E2 -31655.981} C_VEL
LIN {X 0,Y 147.267,Z 815.474,A -85,B 0,C 180,E1 -31655.055,E2 -31655.055} C_VEL
LIN {X 0,Y 136.933,Z 823.345,A -85,B 0,C 180,E1 -31653.917,E2 -31653.917} C_VEL
LIN {X 0,Y 124.926,Z 831.349,A -85,B 0,C 180,E1 -31652.379,E2 -31652.379} C_VEL
LIN {X 0,Y 112.972,Z 838.252,A -85,B 0,C 180,E1 -31650.566,E2 -31650.566} C_VEL
LIN {X 0,Y 102.802,Z 843.369,A -85,B 0,C 180,E1 -31648.709,E2 -31648.709} C_VEL
LIN {X 0,Y 89.469,Z 849.142,A -85,B 0,C 180,E1 -31645.566,E2 -31645.566} C_VEL
LIN {X 0,Y 76.516,Z 853.808,A -85,B 0,C 180,E1 -31641.326,E2 -31641.326} C_VEL
LIN {X 0,Y 61.198,Z 858.237,A -85,B 0,C 180,E1 -31633.553,E2 -31633.553} C_VEL
LIN {X 0,Y 50.237,Z 860.661,A -85,B 0,C 180,E1 -31624.026,E2 -31624.026} C_VEL
LIN {X 0,Y 41.677,Z 862.109,A -85,B 0,C 180,E1 -31609.709,E2 -31609.709} C_VEL
LIN {X 0,Y 37.175,Z 862.641,A -85,B 0,C 180,E1 -31590,E2 -31590} C_VEL
LIN {X 0,Y 41.68,Z 862.109,A -85,B 0,C 180,E1 -31570.292,E2 -31570.292} C_VEL
LIN {X 0,Y 52.331,Z 860.196,A -85,B 0,C 180,E1 -31553.683,E2 -31553.683} C_VEL
LIN {X 0,Y 61.191,Z 858.237,A -85,B 0,C 180,E1 -31546.441,E2 -31546.441} C_VEL
LIN {X 0,Y 76.521,Z 853.807,A -85,B 0,C 180,E1 -31538.679,E2 -31538.679} C_VEL
LIN {X 0,Y 89.468,Z 849.142,A -85,B 0,C 180,E1 -31534.433,E2 -31534.433} C_VEL
LIN {X 0,Y 102.789,Z 843.37,A -85,B 0,C 180,E1 -31531.279,E2 -31531.279} C_VEL
LIN {X 0,Y 116.39,Z 836.432,A -85,B 0,C 180,E1 -31528.885,E2 -31528.885} C_VEL
LIN {X 0,Y 131.812,Z 826.953,A -85,B 0,C 180,E1 -31526.74,E2 -31526.74} C_VEL
LIN {X 0,Y 143.797,Z 818.228,A -85,B 0,C 180,E1 -31525.29,E2 -31525.29} C_VEL
LIN {X 0,Y 154.247,Z 809.645,A -85,B 0,C 180,E1 -31524.322,E2 -31524.322} C_VEL
LIN {X 0,Y 164.681,Z 799.886,A -85,B 0,C 180,E1 -31523.434,E2 -31523.434} C_VEL
LIN {X 0,Y 175.132,Z 788.661,A -85,B 0,C 180,E1 -31522.637,E2 -31522.637} C_VEL
LIN {X 0,Y 180.297,Z 782.518,A -85,B 0,C 180,E1 -31522.228,E2 -31522.228} C_VEL
LIN {X 0,Y 181.998,Z 780.724,A -85,B 0,C 180,E1 -31522.362,E2 -31522.362} C_VEL
LIN {X 0,Y 185.867,Z 789.916,A -85,B 0,C 180,E1 -31530.694,E2 -31530.694} C_VEL
LIN {X 0,Y 195.547,Z 800.036,A -85,B 0,C 180,E1 -31540.309,E2 -31540.309} C_VEL
LIN {X 0,Y 209.445,Z 809.607,A -85,B 0,C 180,E1 -31549.024,E2 -31549.024} C_VEL
LIN {X 0,Y 220.14,Z 816.192,A -85,B 0,C 180,E1 -31554.415,E2 -31554.415} C_VEL
LIN {X 0,Y 229.66,Z 822.427,A -85,B 0,C 180,E1 -31558.963,E2 -31558.963} C_VEL
LIN {X 0,Y 237.311,Z 827.922,A -85,B 0,C 180,E1 -31562.678,E2 -31562.678} C_VEL
LIN {X 0,Y 242.669,Z 831.788,A -85,B 0,C 180,E1 -31565.423,E2 -31565.423} C_VEL
LIN {X 0,Y 247.825,Z 835.479,A -85,B 0,C 180,E1 -31568.367,E2 -31568.367} C_VEL
LIN {X 0,Y 252.364,Z 838.57,A -85,B 0,C 180,E1 -31571.234,E2 -31571.234} C_VEL
LIN {X 0,Y 256.113,Z 841.326,A -85,B 0,C 180,E1 -31574.074,E2 -31574.074} C_VEL
LIN {X 0,Y 259.906,Z 843.939,A -85,B 0,C 180,E1 -31577.507,E2 -31577.507} C_VEL
LIN {X 0,Y 261.591,Z 844.971,A -85,B 0,C 180,E1 -31579.16,E2 -31579.16} C_VEL
LIN {X 0,Y 264.42,Z 846.343,A -85,B 0,C 180,E1 -31582.363,E2 -31582.363} C_VEL
LIN {X 0,Y 265.27,Z 846.763,A -85,B 0,C 180,E1 -31583.643,E2 -31583.643} C_VEL
LIN {X 0,Y 265.448,Z 847.354,A -85,B 0,C 180,E1 -31584.908,E2 -31584.908} C_VEL
LIN {X 0,Y 264.572,Z 848.157,A -85,B 0,C 180,E1 -31586.167,E2 -31586.167} C_VEL
LIN {X 0,Y 260.992,Z 849.956,A -85,B 0,C 180,E1 -31589.57,E2 -31589.57} C_VEL
LIN {X 0,Y 260.648,Z 850.044,A -85,B 0,C 180,E1 -31590.452,E2 -31590.452} C_VEL
LIN {X 0,Y 260.295,Z 849.921,A -85,B 0,C 180,E1 -31592.574,E2 -31592.574} C_VEL
LIN {X 0,Y 259.417,Z 849.581,A -85,B 0,C 180,E1 -31594.662,E2 -31594.662} C_VEL
LIN {X 0,Y 258.59,Z 849.126,A -85,B 0,C 180,E1 -31596.241,E2 -31596.241} C_VEL
LIN {X 0,Y 257.446,Z 848.562,A -85,B 0,C 180,E1 -31597.845,E2 -31597.845} C_VEL
LIN {X 0,Y 254.456,Z 847.013,A -85,B 0,C 180,E1 -31601.147,E2 -31601.147} C_VEL
LIN {X 0,Y 252.476,Z 845.802,A -85,B 0,C 180,E1 -31603.028,E2 -31603.028} C_VEL
LIN {X 0,Y 248.548,Z 843.049,A -85,B 0,C 180,E1 -31606.425,E2 -31606.425} C_VEL
LIN {X 0,Y 245.149,Z 840.607,A -85,B 0,C 180,E1 -31608.908,E2 -31608.908} C_VEL
LIN {X 0,Y 241.345,Z 838.02,A -85,B 0,C 180,E1 -31611.278,E2 -31611.278} C_VEL
LIN {X 0,Y 237.535,Z 835.279,A -85,B 0,C 180,E1 -31613.481,E2 -31613.481} C_VEL
LIN {X 0,Y 231.701,Z 831.099,A -85,B 0,C 180,E1 -31616.521,E2 -31616.521} C_VEL
LIN {X 0,Y 224.664,Z 826.276,A -85,B 0,C 180,E1 -31620.033,E2 -31620.033} C_VEL
LIN {X 0,Y 216.592,Z 821.278,A -85,B 0,C 180,E1 -31623.927,E2 -31623.927} C_VEL
LIN {X 0,Y 207.204,Z 815.585,A -85,B 0,C 180,E1 -31628.73,E2 -31628.73} C_VEL
LIN {X 0,Y 197.131,Z 809.42,A -85,B 0,C 180,E1 -31634.519,E2 -31634.519} C_VEL
LIN {X 0,Y 183.992,Z 799.032,A -85,B 0,C 180,E1 -31645.044,E2 -31645.044} C_VEL
LIN {X 0,Y 177.889,Z 789.092,A -85,B 0,C 180,E1 -31654.873,E2 -31654.873} C_VEL
LIN {X 0,Y 176.435,Z 790.239,A -85,B 0,C 180,E1 -31655.135,E2 -31655.135} C_VEL
LIN {X 0,Y 164.21,Z 803.124,A -85,B 0,C 180,E1 -31653.995,E2 -31653.995} C_VEL
LIN {X 0,Y 152.08,Z 813.971,A -85,B 0,C 180,E1 -31652.727,E2 -31652.727} C_VEL
LIN {X 0,Y 141.91,Z 821.931,A -85,B 0,C 180,E1 -31651.526,E2 -31651.526} C_VEL
LIN {X 0,Y 130.121,Z 830.086,A -85,B 0,C 180,E1 -31649.787,E2 -31649.787} C_VEL
LIN {X 0,Y 116.682,Z 838.042,A -85,B 0,C 180,E1 -31647.483,E2 -31647.483} C_VEL
LIN {X 0,Y 106.729,Z 843.157,A -85,B 0,C 180,E1 -31645.396,E2 -31645.396} C_VEL
LIN {X 0,Y 93.735,Z 848.932,A -85,B 0,C 180,E1 -31641.929,E2 -31641.929} C_VEL
LIN {X 0,Y 81.22,Z 853.598,A -85,B 0,C 180,E1 -31637.349,E2 -31637.349} C_VEL
LIN {X 0,Y 66.614,Z 858.024,A -85,B 0,C 180,E1 -31629.272,E2 -31629.272} C_VEL
LIN {X 0,Y 56.359,Z 860.447,A -85,B 0,C 180,E1 -31619.92,E2 -31619.92} C_VEL
LIN {X 0,Y 48.489,Z 861.895,A -85,B 0,C 180,E1 -31606.85,E2 -31606.85} C_VEL
LIN {X 0,Y 44.336,Z 862.43,A -85,B 0,C 180,E1 -31590,E2 -31590} C_VEL
LIN {X 0,Y 48.491,Z 861.895,A -85,B 0,C 180,E1 -31573.15,E2 -31573.15} C_VEL
LIN {X 0,Y 57.617,Z 860.149,A -85,B 0,C 180,E1 -31558.629,E2 -31558.629} C_VEL
LIN {X 0,Y 66.609,Z 858.024,A -85,B 0,C 180,E1 -31550.724,E2 -31550.724} C_VEL
LIN {X 0,Y 81.225,Z 853.597,A -85,B 0,C 180,E1 -31542.655,E2 -31542.655} C_VEL
LIN {X 0,Y 93.733,Z 848.932,A -85,B 0,C 180,E1 -31538.07,E2 -31538.07} C_VEL
LIN {X 0,Y 106.712,Z 843.158,A -85,B 0,C 180,E1 -31534.591,E2 -31534.591} C_VEL
LIN {X 0,Y 120.665,Z 835.863,A -85,B 0,C 180,E1 -31531.778,E2 -31531.778} C_VEL
LIN {X 0,Y 135.192,Z 826.741,A -85,B 0,C 180,E1 -31529.456,E2 -31529.456} C_VEL
LIN {X 0,Y 147.003,Z 818.02,A -85,B 0,C 180,E1 -31527.818,E2 -31527.818} C_VEL
LIN {X 0,Y 159.066,Z 807.872,A -85,B 0,C 180,E1 -31526.532,E2 -31526.532} C_VEL
LIN {X 0,Y 169.378,Z 797.906,A -85,B 0,C 180,E1 -31525.518,E2 -31525.518} C_VEL
LIN {X 0,Y 176.47,Z 790.251,A -85,B 0,C 180,E1 -31524.901,E2 -31524.901} C_VEL
LIN {X 0,Y 177.883,Z 789.123,A -85,B 0,C 180,E1 -31525.146,E2 -31525.146} C_VEL
LIN {X 0,Y 184.851,Z 799.925,A -85,B 0,C 180,E1 -31535.866,E2 -31535.866} C_VEL
LIN {X 0,Y 198.685,Z 810.445,A -85,B 0,C 180,E1 -31546.479,E2 -31546.479} C_VEL
LIN {X 0,Y 208.873,Z 816.611,A -85,B 0,C 180,E1 -31552.171,E2 -31552.171} C_VEL
LIN {X 0,Y 216.574,Z 821.278,A -85,B 0,C 180,E1 -31556.07,E2 -31556.07} C_VEL
LIN {X 0,Y 224.61,Z 826.278,A -85,B 0,C 180,E1 -31559.959,E2 -31559.959} C_VEL
LIN {X 0,Y 231.7,Z 831.099,A -85,B 0,C 180,E1 -31563.48,E2 -31563.48} C_VEL
LIN {X 0,Y 237.556,Z 835.259,A -85,B 0,C 180,E1 -31566.507,E2 -31566.507} C_VEL
LIN {X 0,Y 242.906,Z 839.09,A -85,B 0,C 180,E1 -31569.685,E2 -31569.685} C_VEL
LIN {X 0,Y 246.07,Z 841.198,A -85,B 0,C 180,E1 -31571.69,E2 -31571.69} C_VEL
LIN {X 0,Y 248.828,Z 843.258,A -85,B 0,C 180,E1 -31573.801,E2 -31573.801} C_VEL
LIN {X 0,Y 252.685,Z 845.93,A -85,B 0,C 180,E1 -31577.144,E2 -31577.144} C_VEL
LIN {X 0,Y 254.433,Z 847.03,A -85,B 0,C 180,E1 -31578.852,E2 -31578.852} C_VEL
LIN {X 0,Y 257.466,Z 848.562,A -85,B 0,C 180,E1 -31582.156,E2 -31582.156} C_VEL
LIN {X 0,Y 258.592,Z 849.138,A -85,B 0,C 180,E1 -31583.759,E2 -31583.759} C_VEL
LIN {X 0,Y 260.111,Z 849.893,A -85,B 0,C 180,E1 -31586.902,E2 -31586.902} C_VEL
LIN {X 0,Y 260.611,Z 850.01,A -85,B 0,C 180,E1 -31588.455,E2 -31588.455} C_VEL
LIN {X 0,Y 260.648,Z 850.044,A -85,B 0,C 180,E1 -31590.452,E2 -31590.452} C_VEL
LIN {X 0,Y 259.794,Z 850.244,A -85,B 0,C 180,E1 -31591.736,E2 -31591.736} C_VEL
LIN {X 0,Y 257.933,Z 850.555,A -85,B 0,C 180,E1 -31592.984,E2 -31592.984} C_VEL
LIN {X 0,Y 253.218,Z 851.091,A -85,B 0,C 180,E1 -31595.472,E2 -31595.472} C_VEL
LIN {X 0,Y 251.366,Z 850.965,A -85,B 0,C 180,E1 -31596.777,E2 -31596.777} C_VEL
LIN {X 0,Y 250.955,Z 850.773,A -85,B 0,C 180,E1 -31597.225,E2 -31597.225} C_VEL
LIN {X 0,Y 248.8,Z 849.675,A -85,B 0,C 180,E1 -31599.758,E2 -31599.758} C_VEL
LIN {X 0,Y 247.118,Z 848.714,A -85,B 0,C 180,E1 -31601.483,E2 -31601.483} C_VEL
LIN {X 0,Y 245.223,Z 847.543,A -85,B 0,C 180,E1 -31603.254,E2 -31603.254} C_VEL
LIN {X 0,Y 241.643,Z 844.992,A -85,B 0,C 180,E1 -31606.308,E2 -31606.308} C_VEL
LIN {X 0,Y 237.893,Z 842.359,A -85,B 0,C 180,E1 -31608.963,E2 -31608.963} C_VEL
LIN {X 0,Y 233.948,Z 839.643,A -85,B 0,C 180,E1 -31611.369,E2 -31611.369} C_VEL
LIN {X 0,Y 230.041,Z 836.841,A -85,B 0,C 180,E1 -31613.577,E2 -31613.577} C_VEL
LIN {X 0,Y 223.952,Z 832.779,A -85,B 0,C 180,E1 -31616.744,E2 -31616.744} C_VEL
LIN {X 0,Y 216.356,Z 827.931,A -85,B 0,C 180,E1 -31620.593,E2 -31620.593} C_VEL
LIN {X 0,Y 206.831,Z 822.393,A -85,B 0,C 180,E1 -31625.364,E2 -31625.364} C_VEL
LIN {X 0,Y 199.362,Z 818.11,A -85,B 0,C 180,E1 -31629.385,E2 -31629.385} C_VEL
LIN {X 0,Y 186.82,Z 810.439,A -85,B 0,C 180,E1 -31637.38,E2 -31637.38} C_VEL
LIN {X 0,Y 175.754,Z 800.098,A -85,B 0,C 180,E1 -31648.679,E2 -31648.679} C_VEL
LIN {X 0,Y 173.941,Z 796.97,A -85,B 0,C 180,E1 -31651.967,E2 -31651.967} C_VEL
LIN {X 0,Y 172.044,Z 798.244,A -85,B 0,C 180,E1 -31652.293,E2 -31652.293} C_VEL
LIN {X 0,Y 160.693,Z 809.223,A -85,B 0,C 180,E1 -31651.008,E2 -31651.008} C_VEL
LIN {X 0,Y 147.11,Z 820.464,A -85,B 0,C 180,E1 -31649.306,E2 -31649.306} C_VEL
LIN {X 0,Y 133.889,Z 829.875,A -85,B 0,C 180,E1 -31647.123,E2 -31647.123} C_VEL
LIN {X 0,Y 120.72,Z 837.832,A -85,B 0,C 180,E1 -31644.59,E2 -31644.59} C_VEL
LIN {X 0,Y 110.979,Z 842.946,A -85,B 0,C 180,E1 -31642.333,E2 -31642.333} C_VEL
LIN {X 0,Y 98.351,Z 848.722,A -85,B 0,C 180,E1 -31638.616,E2 -31638.616} C_VEL
LIN {X 0,Y 86.269,Z 853.387,A -85,B 0,C 180,E1 -31633.824,E2 -31633.824} C_VEL
LIN {X 0,Y 72.365,Z 857.811,A -85,B 0,C 180,E1 -31625.64,E2 -31625.64} C_VEL
LIN {X 0,Y 62.7,Z 860.233,A -85,B 0,C 180,E1 -31616.638,E2 -31616.638} C_VEL
LIN {X 0,Y 55.418,Z 861.681,A -85,B 0,C 180,E1 -31604.692,E2 -31604.692} C_VEL
LIN {X 0,Y 51.487,Z 862.218,A -85,B 0,C 180,E1 -31590,E2 -31590} C_VEL
LIN {X 0,Y 55.42,Z 861.681,A -85,B 0,C 180,E1 -31575.308,E2 -31575.308} C_VEL
LIN {X 0,Y 63.238,Z 860.11,A -85,B 0,C 180,E1 -31562.755,E2 -31562.755} C_VEL
LIN {X 0,Y 72.361,Z 857.811,A -85,B 0,C 180,E1 -31554.357,E2 -31554.357} C_VEL
LIN {X 0,Y 86.273,Z 853.387,A -85,B 0,C 180,E1 -31546.179,E2 -31546.179} C_VEL
LIN {X 0,Y 98.349,Z 848.722,A -85,B 0,C 180,E1 -31541.382,E2 -31541.382} C_VEL
LIN {X 0,Y 110.958,Z 842.947,A -85,B 0,C 180,E1 -31537.654,E2 -31537.654} C_VEL
LIN {X 0,Y 124.191,Z 835.893,A -85,B 0,C 180,E1 -31534.676,E2 -31534.676} C_VEL
LIN {X 0,Y 138.863,Z 826.529,A -85,B 0,C 180,E1 -31532.036,E2 -31532.036} C_VEL
LIN {X 0,Y 150.494,Z 817.811,A -85,B 0,C 180,E1 -31530.241,E2 -31530.241} C_VEL
LIN {X 0,Y 162.404,Z 807.663,A -85,B 0,C 180,E1 -31528.802,E2 -31528.802} C_VEL
LIN {X 0,Y 172.64,Z 797.634,A -85,B 0,C 180,E1 -31527.653,E2 -31527.653} C_VEL
LIN {X 0,Y 173.941,Z 796.977,A -85,B 0,C 180,E1 -31528.037,E2 -31528.037} C_VEL
LIN {X 0,Y 181.6,Z 806.413,A -85,B 0,C 180,E1 -31538.257,E2 -31538.257} C_VEL
LIN {X 0,Y 192.849,Z 814.357,A -85,B 0,C 180,E1 -31546.79,E2 -31546.79} C_VEL
LIN {X 0,Y 203.167,Z 820.329,A -85,B 0,C 180,E1 -31552.713,E2 -31552.713} C_VEL
LIN {X 0,Y 210.577,Z 824.61,A -85,B 0,C 180,E1 -31556.55,E2 -31556.55} C_VEL
LIN {X 0,Y 218.288,Z 829.156,A -85,B 0,C 180,E1 -31560.375,E2 -31560.375} C_VEL
LIN {X 0,Y 226.103,Z 834.18,A -85,B 0,C 180,E1 -31564.343,E2 -31564.343} C_VEL
LIN {X 0,Y 232.013,Z 838.23,A -85,B 0,C 180,E1 -31567.497,E2 -31567.497} C_VEL
LIN {X 0,Y 236.235,Z 841.201,A -85,B 0,C 180,E1 -31569.995,E2 -31569.995} C_VEL
LIN {X 0,Y 239.495,Z 843.395,A -85,B 0,C 180,E1 -31572.054,E2 -31572.054} C_VEL
LIN {X 0,Y 243.125,Z 846.086,A -85,B 0,C 180,E1 -31574.921,E2 -31574.921} C_VEL
LIN {X 0,Y 245.378,Z 847.638,A -85,B 0,C 180,E1 -31576.856,E2 -31576.856} C_VEL
LIN {X 0,Y 248.794,Z 849.69,A -85,B 0,C 180,E1 -31580.242,E2 -31580.242} C_VEL
LIN {X 0,Y 250.348,Z 850.466,A -85,B 0,C 180,E1 -31581.931,E2 -31581.931} C_VEL
LIN {X 0,Y 251.608,Z 851.102,A -85,B 0,C 180,E1 -31583.585,E2 -31583.585} C_VEL
LIN {X 0,Y 252.513,Z 851.567,A -85,B 0,C 180,E1 -31585.211,E2 -31585.211} C_VEL
LIN {X 0,Y 253.342,Z 851.865,A -85,B 0,C 180,E1 -31587.041,E2 -31587.041} C_VEL
LIN {X 0,Y 253.764,Z 851.989,A -85,B 0,C 180,E1 -31588.413,E2 -31588.413} C_VEL
LIN {X 0,Y 253.834,Z 852.025,A -85,B 0,C 180,E1 -31590.411,E2 -31590.411} C_VEL
LIN {X 0,Y 253.34,Z 851.847,A -85,B 0,C 180,E1 -31592.95,E2 -31592.95} C_VEL
LIN {X 0,Y 252.513,Z 851.541,A -85,B 0,C 180,E1 -31594.789,E2 -31594.789} C_VEL
LIN {X 0,Y 250.955,Z 850.773,A -85,B 0,C 180,E1 -31597.225,E2 -31597.225} C_VEL
LIN {X 0,Y 249.259,Z 850.443,A -85,B 0,C 180,E1 -31598.515,E2 -31598.515} C_VEL
LIN {X 0,Y 246.611,Z 850.269,A -85,B 0,C 180,E1 -31599.743,E2 -31599.743} C_VEL
LIN {X 0,Y 240.461,Z 849.666,A -85,B 0,C 180,E1 -31602.173,E2 -31602.173} C_VEL
LIN {X 0,Y 237.942,Z 848.905,A -85,B 0,C 180,E1 -31603.469,E2 -31603.469} C_VEL
LIN {X 0,Y 237.318,Z 848.55,A -85,B 0,C 180,E1 -31603.92,E2 -31603.92} C_VEL
LIN {X 0,Y 234.378,Z 846.419,A -85,B 0,C 180,E1 -31606.356,E2 -31606.356} C_VEL
LIN {X 0,Y 232.755,Z 845.228,A -85,B 0,C 180,E1 -31607.574,E2 -31607.574} C_VEL
LIN {X 0,Y 229.38,Z 842.946,A -85,B 0,C 180,E1 -31609.696,E2 -31609.696} C_VEL
LIN {X 0,Y 225.585,Z 840.317,A -85,B 0,C 180,E1 -31611.953,E2 -31611.953} C_VEL
LIN {X 0,Y 221.131,Z 837.439,A -85,B 0,C 180,E1 -31614.403,E2 -31614.403} C_VEL
LIN {X 0,Y 212.599,Z 832.231,A -85,B 0,C 180,E1 -31618.835,E2 -31618.835} C_VEL
LIN {X 0,Y 206.719,Z 828.965,A -85,B 0,C 180,E1 -31621.796,E2 -31621.796} C_VEL
LIN {X 0,Y 199.159,Z 824.843,A -85,B 0,C 180,E1 -31625.746,E2 -31625.746} C_VEL
LIN {X 0,Y 188.593,Z 819.07,A -85,B 0,C 180,E1 -31631.816,E2 -31631.816} C_VEL
LIN {X 0,Y 174.659,Z 809.551,A -85,B 0,C 180,E1 -31642.875,E2 -31642.875} C_VEL
LIN {X 0,Y 169.94,Z 804.111,A -85,B 0,C 180,E1 -31649.247,E2 -31649.247} C_VEL
LIN {X 0,Y 168.296,Z 805.274,A -85,B 0,C 180,E1 -31649.336,E2 -31649.336} C_VEL
LIN {X 0,Y 157.612,Z 814.846,A -85,B 0,C 180,E1 -31647.908,E2 -31647.908} C_VEL
LIN {X 0,Y 146.024,Z 823.926,A -85,B 0,C 180,E1 -31646.12,E2 -31646.12} C_VEL
LIN {X 0,Y 134.674,Z 831.77,A -85,B 0,C 180,E1 -31643.984,E2 -31643.984} C_VEL
LIN {X 0,Y 121.849,Z 839.438,A -85,B 0,C 180,E1 -31641.136,E2 -31641.136} C_VEL
LIN {X 0,Y 106.291,Z 847.206,A -85,B 0,C 180,E1 -31636.661,E2 -31636.661} C_VEL
LIN {X 0,Y 94.499,Z 852.132,A -85,B 0,C 180,E1 -31632.015,E2 -31632.015} C_VEL
LIN {X 0,Y 83.462,Z 855.987,A -85,B 0,C 180,E1 -31626.116,E2 -31626.116} C_VEL
LIN {X 0,Y 73.579,Z 858.881,A -85,B 0,C 180,E1 -31618.527,E2 -31618.527} C_VEL
LIN {X 0,Y 65.482,Z 860.81,A -85,B 0,C 180,E1 -31608.782,E2 -31608.782} C_VEL
LIN {X 0,Y 60.092,Z 861.787,A -85,B 0,C 180,E1 -31596.716,E2 -31596.716} C_VEL
LIN {X 0,Y 58.63,Z 862.007,A -85,B 0,C 180,E1 -31590,E2 -31590} C_VEL
LIN {X 0,Y 62.402,Z 861.467,A -85,B 0,C 180,E1 -31576.983,E2 -31576.983} C_VEL
LIN {X 0,Y 69.249,Z 860.017,A -85,B 0,C 180,E1 -31566.05,E2 -31566.05} C_VEL
LIN {X 0,Y 78.345,Z 857.599,A -85,B 0,C 180,E1 -31557.437,E2 -31557.437} C_VEL
LIN {X 0,Y 91.617,Z 853.177,A -85,B 0,C 180,E1 -31549.305,E2 -31549.305} C_VEL
LIN {X 0,Y 103.265,Z 848.511,A -85,B 0,C 180,E1 -31544.39,E2 -31544.39} C_VEL
LIN {X 0,Y 115.513,Z 842.735,A -85,B 0,C 180,E1 -31540.492,E2 -31540.492} C_VEL
LIN {X 0,Y 129.656,Z 834.934,A -85,B 0,C 180,E1 -31537.046,E2 -31537.046} C_VEL
LIN {X 0,Y 142.817,Z 826.316,A -85,B 0,C 180,E1 -31534.488,E2 -31534.488} C_VEL
LIN {X 0,Y 154.248,Z 817.602,A -85,B 0,C 180,E1 -31532.553,E2 -31532.553} C_VEL
LIN {X 0,Y 165.703,Z 807.712,A -85,B 0,C 180,E1 -31531.008,E2 -31531.008} C_VEL
LIN {X 0,Y 168.307,Z 805.272,A -85,B 0,C 180,E1 -31530.669,E2 -31530.669} C_VEL
LIN {X 0,Y 169.955,Z 804.111,A -85,B 0,C 180,E1 -31530.762,E2 -31530.762} C_VEL
LIN {X 0,Y 180.048,Z 813.771,A -85,B 0,C 180,E1 -31542.13,E2 -31542.13} C_VEL
LIN {X 0,Y 191.957,Z 820.968,A -85,B 0,C 180,E1 -31550.25,E2 -31550.25} C_VEL
LIN {X 0,Y 199.154,Z 824.849,A -85,B 0,C 180,E1 -31554.256,E2 -31554.256} C_VEL
LIN {X 0,Y 206.716,Z 828.968,A -85,B 0,C 180,E1 -31558.206,E2 -31558.206} C_VEL
LIN {X 0,Y 212.578,Z 832.255,A -85,B 0,C 180,E1 -31561.175,E2 -31561.175} C_VEL
LIN {X 0,Y 218.504,Z 835.812,A -85,B 0,C 180,E1 -31564.235,E2 -31564.235} C_VEL
LIN {X 0,Y 222.524,Z 838.32,A -85,B 0,C 180,E1 -31566.333,E2 -31566.333} C_VEL
LIN {X 0,Y 226.491,Z 840.958,A -85,B 0,C 180,E1 -31568.573,E2 -31568.573} C_VEL
LIN {X 0,Y 230.472,Z 843.682,A -85,B 0,C 180,E1 -31570.961,E2 -31570.961} C_VEL
LIN {X 0,Y 232.79,Z 845.221,A -85,B 0,C 180,E1 -31572.429,E2 -31572.429} C_VEL
LIN {X 0,Y 235.368,Z 847.138,A -85,B 0,C 180,E1 -31574.411,E2 -31574.411} C_VEL
LIN {X 0,Y 238.199,Z 849.129,A -85,B 0,C 180,E1 -31576.816,E2 -31576.816} C_VEL
LIN {X 0,Y 241.456,Z 851.164,A -85,B 0,C 180,E1 -31579.943,E2 -31579.943} C_VEL
LIN {X 0,Y 243.107,Z 852.032,A -85,B 0,C 180,E1 -31581.689,E2 -31581.689} C_VEL
LIN {X 0,Y 244.486,Z 852.683,A -85,B 0,C 180,E1 -31583.397,E2 -31583.397} C_VEL
LIN {X 0,Y 245.49,Z 853.168,A -85,B 0,C 180,E1 -31585.073,E2 -31585.073} C_VEL
LIN {X 0,Y 246.338,Z 853.52,A -85,B 0,C 180,E1 -31586.895,E2 -31586.895} C_VEL
LIN {X 0,Y 246.831,Z 853.665,A -85,B 0,C 180,E1 -31588.368,E2 -31588.368} C_VEL
LIN {X 0,Y 246.994,Z 853.722,A -85,B 0,C 180,E1 -31590,E2 -31590} C_VEL
LIN {X 0,Y 246.803,Z 853.661,A -85,B 0,C 180,E1 -31591.632,E2 -31591.632} C_VEL
LIN {X 0,Y 246.25,Z 853.481,A -85,B 0,C 180,E1 -31593.272,E2 -31593.272} C_VEL
LIN {X 0,Y 245.488,Z 853.146,A -85,B 0,C 180,E1 -31594.927,E2 -31594.927} C_VEL
LIN {X 0,Y 244.156,Z 852.53,A -85,B 0,C 180,E1 -31596.957,E2 -31596.957} C_VEL
LIN {X 0,Y 242.166,Z 851.513,A -85,B 0,C 180,E1 -31599.35,E2 -31599.35} C_VEL
LIN {X 0,Y 239.651,Z 850.087,A -85,B 0,C 180,E1 -31601.846,E2 -31601.846} C_VEL
LIN {X 0,Y 237.318,Z 848.55,A -85,B 0,C 180,E1 -31603.92,E2 -31603.92} C_VEL
LIN {X 0,Y 235.912,Z 847.916,A -85,B 0,C 180,E1 -31604.792,E2 -31604.792} C_VEL
LIN {X 0,Y 232.929,Z 847.071,A -85,B 0,C 180,E1 -31606.025,E2 -31606.025} C_VEL
LIN {X 0,Y 222.316,Z 844.145,A -85,B 0,C 180,E1 -31609.637,E2 -31609.637} C_VEL
LIN {X 0,Y 220.517,Z 843.221,A -85,B 0,C 180,E1 -31610.538,E2 -31610.538} C_VEL
LIN {X 0,Y 214.95,Z 839.751,A -85,B 0,C 180,E1 -31613.727,E2 -31613.727} C_VEL
LIN {X 0,Y 206.907,Z 835.213,A -85,B 0,C 180,E1 -31617.978,E2 -31617.978} C_VEL
LIN {X 0,Y 198.986,Z 831.097,A -85,B 0,C 180,E1 -31622.044,E2 -31622.044} C_VEL
LIN {X 0,Y 191.429,Z 827.197,A -85,B 0,C 180,E1 -31626.13,E2 -31626.13} C_VEL
LIN {X 0,Y 180.997,Z 821.756,A -85,B 0,C 180,E1 -31632.46,E2 -31632.46} C_VEL
LIN {X 0,Y 167.725,Z 812.589,A -85,B 0,C 180,E1 -31644.083,E2 -31644.083} C_VEL
LIN {X 0,Y 166.36,Z 811.121,A -85,B 0,C 180,E1 -31645.962,E2 -31645.962} C_VEL
LIN {X 0,Y 163.782,Z 812.719,A -85,B 0,C 180,E1 -31646.094,E2 -31646.094} C_VEL
LIN {X 0,Y 151.718,Z 822.512,A -85,B 0,C 180,E1 -31644.157,E2 -31644.157} C_VEL
LIN {X 0,Y 140.618,Z 830.509,A -85,B 0,C 180,E1 -31641.92,E2 -31641.92} C_VEL
LIN {X 0,Y 129.455,Z 837.502,A -85,B 0,C 180,E1 -31639.349,E2 -31639.349} C_VEL
LIN {X 0,Y 117.331,Z 844.068,A -85,B 0,C 180,E1 -31635.953,E2 -31635.953} C_VEL
LIN {X 0,Y 105.552,Z 849.59,A -85,B 0,C 180,E1 -31631.745,E2 -31631.745} C_VEL
LIN {X 0,Y 94.541,Z 853.997,A -85,B 0,C 180,E1 -31626.491,E2 -31626.491} C_VEL
LIN {X 0,Y 84.528,Z 857.386,A -85,B 0,C 180,E1 -31619.924,E2 -31619.924} C_VEL
LIN {X 0,Y 75.239,Z 859.962,A -85,B 0,C 180,E1 -31610.922,E2 -31610.922} C_VEL
LIN {X 0,Y 69.418,Z 861.253,A -85,B 0,C 180,E1 -31601.682,E2 -31601.682} C_VEL
LIN {X 0,Y 65.806,Z 861.795,A -85,B 0,C 180,E1 -31590,E2 -31590} C_VEL
LIN {X 0,Y 69.419,Z 861.253,A -85,B 0,C 180,E1 -31578.318,E2 -31578.318} C_VEL
LIN {X 0,Y 75.907,Z 859.802,A -85,B 0,C 180,E1 -31568.263,E2 -31568.263} C_VEL
LIN {X 0,Y 84.526,Z 857.386,A -85,B 0,C 180,E1 -31560.075,E2 -31560.075} C_VEL
LIN {X 0,Y 94.545,Z 853.996,A -85,B 0,C 180,E1 -31553.511,E2 -31553.511} C_VEL
LIN {X 0,Y 105.55,Z 849.59,A -85,B 0,C 180,E1 -31548.254,E2 -31548.254} C_VEL
LIN {X 0,Y 117.309,Z 844.069,A -85,B 0,C 180,E1 -31544.036,E2 -31544.036} C_VEL
LIN {X 0,Y 129.608,Z 837.413,A -85,B 0,C 180,E1 -31540.612,E2 -31540.612} C_VEL
LIN {X 0,Y 142.222,Z 829.45,A -85,B 0,C 180,E1 -31537.756,E2 -31537.756} C_VEL
LIN {X 0,Y 154.962,Z 820.035,A -85,B 0,C 180,E1 -31535.28,E2 -31535.28} C_VEL
LIN {X 0,Y 163.783,Z 812.719,A -85,B 0,C 180,E1 -31533.905,E2 -31533.905} C_VEL
LIN {X 0,Y 166.361,Z 811.12,A -85,B 0,C 180,E1 -31534.038,E2 -31534.038} C_VEL
LIN {X 0,Y 177.854,Z 820.019,A -85,B 0,C 180,E1 -31545.338,E2 -31545.338} C_VEL
LIN {X 0,Y 187.79,Z 825.411,A -85,B 0,C 180,E1 -31551.805,E2 -31551.805} C_VEL
LIN {X 0,Y 195.163,Z 829.11,A -85,B 0,C 180,E1 -31555.918,E2 -31555.918} C_VEL
